LIN {X 0,Y 441.161,Z 147.091,A -85,B 0,C 180,E1 16742.338,E2 16742.338} C_VEL
LIN {X 0,Y 441.166,Z 147.092,A -85,B 0,C 180,E1 16738.571,E2 16738.571} C_VEL
LIN {X 0,Y 441.182,Z 147.089,A -85,B 0,C 180,E1 16734.929,E2 16734.929} C_VEL
LIN {X 0,Y 441.199,Z 147.088,A -85,B 0,C 180,E1 16731.266,E2 16731.266} C_VEL
LIN {X 0,Y 441.19,Z 147.092,A -85,B 0,C 180,E1 16727.434,E2 16727.434} C_VEL
LIN {X 0,Y 441.161,Z 147.096,A -85,B 0,C 180,E1 16723.813,E2 16723.813} C_VEL
LIN {X 0,Y 441.139,Z 147.048,A -85,B 0,C 180,E1 16720.124,E2 16720.124} C_VEL
LIN {X 0,Y 441.139,Z 147.074,A -85,B 0,C 180,E1 16716.348,E2 16716.348} C_VEL
LIN {X 0,Y 441.143,Z 147.081,A -85,B 0,C 180,E1 16712.606,E2 16712.606} C_VEL
LIN {X 0,Y 441.168,Z 147.048,A -85,B 0,C 180,E1 16709.038,E2 16709.038} C_VEL
LIN {X 0,Y 441.209,Z 147.301,A -85,B 0,C 180,E1 16705.273,E2 16705.273} C_VEL
LIN {X 0,Y 442.541,Z 150.696,A -85,B 0,C 180,E1 16704.503,E2 16704.503} C_VEL
LIN {X 0,Y 444.11,Z 153.026,A -85,B 0,C 180,E1 16703.923,E2 16703.923} C_VEL
LIN {X 0,Y 446.863,Z 158.227,A -85,B 0,C 180,E1 16702.8,E2 16702.8} C_VEL
LIN {X 0,Y 449.775,Z 163.654,A -85,B 0,C 180,E1 16701.667,E2 16701.667} C_VEL
LIN {X 0,Y 455.654,Z 174.722,A -85,B 0,C 180,E1 16699.494,E2 16699.494} C_VEL
LIN {X 0,Y 463.787,Z 191.79,A -85,B 0,C 180,E1 16696.55,E2 16696.55} C_VEL
LIN {X 0,Y 469.472,Z 204.192,A -85,B 0,C 180,E1 16694.656,E2 16694.656} C_VEL
LIN {X 0,Y 470.709,Z 206.682,A -85,B 0,C 180,E1 16694.44,E2 16694.44} C_VEL
LIN {X 0,Y 475.94,Z 241.296,A -85,B 0,C 180,E1 16693.055,E2 16693.055} C_VEL
LIN {X 0,Y 471.437,Z 427.319,A -85,B 0,C 180,E1 16689.939,E2 16689.939} C_VEL
LIN {X 0,Y 470.53,Z 435.022,A -85,B 0,C 180,E1 16689.894,E2 16689.894} C_VEL
LIN {X 0,Y 465.461,Z 455.605,A -85,B 0,C 180,E1 16690.074,E2 16690.074} C_VEL
LIN {X 0,Y 464.744,Z 462.217,A -85,B 0,C 180,E1 16690.028,E2 16690.028} C_VEL
LIN {X 0,Y 463.247,Z 517.307,A -85,B 0,C 180,E1 16689.082,E2 16689.082} C_VEL
LIN {X 0,Y 461.864,Z 538.343,A -85,B 0,C 180,E1 16688.519,E2 16688.519} C_VEL
LIN {X 0,Y 459.97,Z 559.929,A -85,B 0,C 180,E1 16687.719,E2 16687.719} C_VEL
LIN {X 0,Y 457.77,Z 579.888,A -85,B 0,C 180,E1 16686.759,E2 16686.759} C_VEL
LIN {X 0,Y 455.2,Z 599.112,A -85,B 0,C 180,E1 16685.596,E2 16685.596} C_VEL
LIN {X 0,Y 452.431,Z 617.858,A -85,B 0,C 180,E1 16684.223,E2 16684.223} C_VEL
LIN {X 0,Y 449.568,Z 634.992,A -85,B 0,C 180,E1 16682.713,E2 16682.713} C_VEL
LIN {X 0,Y 446.418,Z 652.781,A -85,B 0,C 180,E1 16680.856,E2 16680.856} C_VEL
LIN {X 0,Y 443.483,Z 669.165,A -85,B 0,C 180,E1 16678.846,E2 16678.846} C_VEL
LIN {X 0,Y 440.701,Z 684.442,A -85,B 0,C 180,E1 16676.632,E2 16676.632} C_VEL
LIN {X 0,Y 438.261,Z 698.588,A -85,B 0,C 180,E1 16674.245,E2 16674.245} C_VEL
LIN {X 0,Y 436.194,Z 711.687,A -85,B 0,C 180,E1 16671.656,E2 16671.656} C_VEL
LIN {X 0,Y 434.567,Z 723.315,A -85,B 0,C 180,E1 16668.93,E2 16668.93} C_VEL
LIN {X 0,Y 433.412,Z 732.998,A -85,B 0,C 180,E1 16666.208,E2 16666.208} C_VEL
LIN {X 0,Y 432.635,Z 741.395,A -85,B 0,C 180,E1 16663.351,E2 16663.351} C_VEL
LIN {X 0,Y 432.205,Z 748.037,A -85,B 0,C 180,E1 16660.519,E2 16660.519} C_VEL
LIN {X 0,Y 431.991,Z 753.036,A -85,B 0,C 180,E1 16657.715,E2 16657.715} C_VEL
LIN {X 0,Y 431.924,Z 756.563,A -85,B 0,C 180,E1 16654.913,E2 16654.913} C_VEL
LIN {X 0,Y 431.907,Z 758.422,A -85,B 0,C 180,E1 16652.255,E2 16652.255} C_VEL
LIN {X 0,Y 431.902,Z 758.898,A -85,B 0,C 180,E1 16649.337,E2 16649.337} C_VEL
LIN {X 0,Y 431.914,Z 757.928,A -85,B 0,C 180,E1 16646.682,E2 16646.682} C_VEL
LIN {X 0,Y 431.947,Z 755.334,A -85,B 0,C 180,E1 16643.888,E2 16643.888} C_VEL
LIN {X 0,Y 432.054,Z 751.256,A -85,B 0,C 180,E1 16641.08,E2 16641.08} C_VEL
LIN {X 0,Y 432.365,Z 745.257,A -85,B 0,C 180,E1 16638.123,E2 16638.123} C_VEL
LIN {X 0,Y 432.935,Z 737.852,A -85,B 0,C 180,E1 16635.283,E2 16635.283} C_VEL
LIN {X 0,Y 433.837,Z 729.193,A -85,B 0,C 180,E1 16632.566,E2 16632.566} C_VEL
LIN {X 0,Y 435.177,Z 718.684,A -85,B 0,C 180,E1 16629.841,E2 16629.841} C_VEL
LIN {X 0,Y 436.927,Z 706.823,A -85,B 0,C 180,E1 16627.249,E2 16627.249} C_VEL
LIN {X 0,Y 439.099,Z 693.731,A -85,B 0,C 180,E1 16624.799,E2 16624.799} C_VEL
LIN {X 0,Y 441.803,Z 678.428,A -85,B 0,C 180,E1 16622.359,E2 16622.359} C_VEL
LIN {X 0,Y 444.668,Z 662.439,A -85,B 0,C 180,E1 16620.204,E2 16620.204} C_VEL
LIN {X 0,Y 447.82,Z 645.002,A -85,B 0,C 180,E1 16618.203,E2 16618.203} C_VEL
LIN {X 0,Y 450.894,Z 627.379,A -85,B 0,C 180,E1 16616.486,E2 16616.486} C_VEL
LIN {X 0,Y 453.696,Z 609.476,A -85,B 0,C 180,E1 16615.042,E2 16615.042} C_VEL
LIN {X 0,Y 456.596,Z 589.037,A -85,B 0,C 180,E1 16613.678,E2 16613.678} C_VEL
LIN {X 0,Y 459.081,Z 568.729,A -85,B 0,C 180,E1 16612.581,E2 16612.581} C_VEL
LIN {X 0,Y 461.105,Z 547.553,A -85,B 0,C 180,E1 16611.7,E2 16611.7} C_VEL
LIN {X 0,Y 462.765,Z 525.423,A -85,B 0,C 180,E1 16611.024,E2 16611.024} C_VEL
LIN {X 0,Y 463.781,Z 503.548,A -85,B 0,C 180,E1 16610.568,E2 16610.568} C_VEL
LIN {X 0,Y 469.385,Z 276.561,A -85,B 0,C 180,E1 16606.757,E2 16606.757} C_VEL
LIN {X 0,Y 470.228,Z 241.192,A -85,B 0,C 180,E1 16606.129,E2 16606.129} C_VEL
LIN {X 0,Y 465.388,Z 210.155,A -85,B 0,C 180,E1 16604.831,E2 16604.831} C_VEL
LIN {X 0,Y 460.669,Z 202.535,A -85,B 0,C 180,E1 16603.991,E2 16603.991} C_VEL
LIN {X 0,Y 453.502,Z 187.149,A -85,B 0,C 180,E1 16601.409,E2 16601.409} C_VEL
LIN {X 0,Y 447.296,Z 174.728,A -85,B 0,C 180,E1 16599.077,E2 16599.077} C_VEL
LIN {X 0,Y 442.959,Z 166.509,A -85,B 0,C 180,E1 16597.387,E2 16597.387} C_VEL
LIN {X 0,Y 440.374,Z 161.697,A -85,B 0,C 180,E1 16596.341,E2 16596.341} C_VEL
LIN {X 0,Y 438.184,Z 157.597,A -85,B 0,C 180,E1 16595.421,E2 16595.421} C_VEL
LIN {X 0,Y 436.317,Z 154.259,A -85,B 0,C 180,E1 16594.633,E2 16594.633} C_VEL
LIN {X 0,Y 435.776,Z 153.005,A -85,B 0,C 180,E1 16594.363,E2 16594.363} C_VEL
LIN {X 0,Y 433.766,Z 150.233,A -85,B 0,C 180,E1 16593.588,E2 16593.588} C_VEL
LIN {X 0,Y 433.233,Z 148.247,A -85,B 0,C 180,E1 16593.097,E2 16593.097} C_VEL
LIN {X 0,Y 433.191,Z 148.054,A -85,B 0,C 180,E1 16589.525,E2 16589.525} C_VEL
LIN {X 0,Y 433.19,Z 148.038,A -85,B 0,C 180,E1 16585.717,E2 16585.717} C_VEL
LIN {X 0,Y 433.201,Z 148.086,A -85,B 0,C 180,E1 16581.903,E2 16581.903} C_VEL
LIN {X 0,Y 433.209,Z 148.039,A -85,B 0,C 180,E1 16578.155,E2 16578.155} C_VEL
LIN {X 0,Y 433.236,Z 148.069,A -85,B 0,C 180,E1 16574.433,E2 16574.433} C_VEL
LIN {X 0,Y 433.248,Z 148.069,A -85,B 0,C 180,E1 16570.639,E2 16570.639} C_VEL
LIN {X 0,Y 433.265,Z 148.068,A -85,B 0,C 180,E1 16566.759,E2 16566.759} C_VEL
LIN {X 0,Y 433.248,Z 148.072,A -85,B 0,C 180,E1 16562.91,E2 16562.91} C_VEL
LIN {X 0,Y 433.234,Z 148.075,A -85,B 0,C 180,E1 16559.207,E2 16559.207} C_VEL
LIN {X 0,Y 433.224,Z 148.079,A -85,B 0,C 180,E1 16555.5,E2 16555.5} C_VEL
LIN {X 0,Y 433.224,Z 148.08,A -85,B 0,C 180,E1 16551.773,E2 16551.773} C_VEL
LIN {X 0,Y 433.233,Z 148.08,A -85,B 0,C 180,E1 16548.012,E2 16548.012} C_VEL
LIN {X 0,Y 433.239,Z 148.026,A -85,B 0,C 180,E1 16544.228,E2 16544.228} C_VEL
LIN {X 0,Y 433.256,Z 148.061,A -85,B 0,C 180,E1 16540.45,E2 16540.45} C_VEL
LIN {X 0,Y 433.257,Z 148.052,A -85,B 0,C 180,E1 16536.613,E2 16536.613} C_VEL
LIN {X 0,Y 433.251,Z 148.032,A -85,B 0,C 180,E1 16532.81,E2 16532.81} C_VEL
LIN {X 0,Y 433.288,Z 148.284,A -85,B 0,C 180,E1 16529.184,E2 16529.184} C_VEL
LIN {X 0,Y 434.702,Z 151.729,A -85,B 0,C 180,E1 16528.371,E2 16528.371} C_VEL
LIN {X 0,Y 436.151,Z 153.411,A -85,B 0,C 180,E1 16527.87,E2 16527.87} C_VEL
LIN {X 0,Y 437.891,Z 157.074,A -85,B 0,C 180,E1 16527.082,E2 16527.082} C_VEL
LIN {X 0,Y 439.231,Z 159.208,A -85,B 0,C 180,E1 16526.573,E2 16526.573} C_VEL
LIN {X 0,Y 444.555,Z 168.866,A -85,B 0,C 180,E1 16524.504,E2 16524.504} C_VEL
LIN {X 0,Y 452.392,Z 179.593,A -85,B 0,C 180,E1 16522.928,E2 16522.928} C_VEL
LIN {X 0,Y 462.317,Z 193.566,A -85,B 0,C 180,E1 16521.134,E2 16521.134} C_VEL
LIN {X 0,Y 474.451,Z 211.926,A -85,B 0,C 180,E1 16519.09,E2 16519.09} C_VEL
LIN {X 0,Y 474.756,Z 213.111,A -85,B 0,C 180,E1 16519.025,E2 16519.025} C_VEL
LIN {X 0,Y 467.958,Z 425.301,A -85,B 0,C 180,E1 16515.184,E2 16515.184} C_VEL
LIN {X 0,Y 465.168,Z 512.028,A -85,B 0,C 180,E1 16513.602,E2 16513.602} C_VEL
LIN {X 0,Y 463.607,Z 534.936,A -85,B 0,C 180,E1 16512.987,E2 16512.987} C_VEL
LIN {X 0,Y 461.686,Z 557.609,A -85,B 0,C 180,E1 16512.17,E2 16512.17} C_VEL
LIN {X 0,Y 459.492,Z 578.606,A -85,B 0,C 180,E1 16511.197,E2 16511.197} C_VEL
LIN {X 0,Y 456.901,Z 600.642,A -85,B 0,C 180,E1 16509.961,E2 16509.961} C_VEL
LIN {X 0,Y 454.323,Z 620.398,A -85,B 0,C 180,E1 16508.623,E2 16508.623} C_VEL
LIN {X 0,Y 451.294,Z 641.976,A -85,B 0,C 180,E1 16506.888,E2 16506.888} C_VEL
LIN {X 0,Y 448.466,Z 660.864,A -85,B 0,C 180,E1 16505.113,E2 16505.113} C_VEL
LIN {X 0,Y 445.625,Z 678.963,A -85,B 0,C 180,E1 16503.116,E2 16503.116} C_VEL
LIN {X 0,Y 442.903,Z 696.137,A -85,B 0,C 180,E1 16500.924,E2 16500.924} C_VEL
LIN {X 0,Y 440.427,Z 711.612,A -85,B 0,C 180,E1 16498.62,E2 16498.62} C_VEL
LIN {X 0,Y 438.093,Z 726.942,A -85,B 0,C 180,E1 16495.988,E2 16495.988} C_VEL
LIN {X 0,Y 436.406,Z 738.708,A -85,B 0,C 180,E1 16493.637,E2 16493.637} C_VEL
LIN {X 0,Y 434.67,Z 751.426,A -85,B 0,C 180,E1 16490.576,E2 16490.576} C_VEL
LIN {X 0,Y 433.525,Z 761.436,A -85,B 0,C 180,E1 16487.724,E2 16487.724} C_VEL
LIN {X 0,Y 432.749,Z 769.699,A -85,B 0,C 180,E1 16484.86,E2 16484.86} C_VEL
LIN {X 0,Y 432.293,Z 776.47,A -85,B 0,C 180,E1 16482.014,E2 16482.014} C_VEL
LIN {X 0,Y 432.033,Z 781.843,A -85,B 0,C 180,E1 16479.054,E2 16479.054} C_VEL
LIN {X 0,Y 431.943,Z 785.438,A -85,B 0,C 180,E1 16476.379,E2 16476.379} C_VEL
LIN {X 0,Y 431.91,Z 787.984,A -85,B 0,C 180,E1 16473.318,E2 16473.318} C_VEL
LIN {X 0,Y 431.901,Z 788.894,A -85,B 0,C 180,E1 16470.663,E2 16470.663} C_VEL
LIN {X 0,Y 431.907,Z 788.46,A -85,B 0,C 180,E1 16467.612,E2 16467.612} C_VEL
LIN {X 0,Y 431.919,Z 786.727,A -85,B 0,C 180,E1 16464.953,E2 16464.953} C_VEL
LIN {X 0,Y 431.998,Z 783.494,A -85,B 0,C 180,E1 16462.018,E2 16462.018} C_VEL
LIN {X 0,Y 432.177,Z 778.573,A -85,B 0,C 180,E1 16459.064,E2 16459.064} C_VEL
LIN {X 0,Y 432.574,Z 772.169,A -85,B 0,C 180,E1 16456.091,E2 16456.091} C_VEL
LIN {X 0,Y 433.216,Z 764.337,A -85,B 0,C 180,E1 16453.232,E2 16453.232} C_VEL
LIN {X 0,Y 434.298,Z 754.411,A -85,B 0,C 180,E1 16450.219,E2 16450.219} C_VEL
LIN {X 0,Y 435.626,Z 744.143,A -85,B 0,C 180,E1 16447.605,E2 16447.605} C_VEL
LIN {X 0,Y 437.263,Z 732.76,A -85,B 0,C 180,E1 16445.119,E2 16445.119} C_VEL
LIN {X 0,Y 439.298,Z 718.902,A -85,B 0,C 180,E1 16442.579,E2 16442.579} C_VEL
LIN {X 0,Y 441.866,Z 702.557,A -85,B 0,C 180,E1 16439.996,E2 16439.996} C_VEL
LIN {X 0,Y 444.462,Z 686.329,A -85,B 0,C 180,E1 16437.782,E2 16437.782} C_VEL
LIN {X 0,Y 447.256,Z 668.628,A -85,B 0,C 180,E1 16435.713,E2 16435.713} C_VEL
LIN {X 0,Y 450.17,Z 649.602,A -85,B 0,C 180,E1 16433.787,E2 16433.787} C_VEL
LIN {X 0,Y 453.07,Z 629.567,A -85,B 0,C 180,E1 16432.078,E2 16432.078} C_VEL
LIN {X 0,Y 455.981,Z 608.032,A -85,B 0,C 180,E1 16430.514,E2 16430.514} C_VEL
LIN {X 0,Y 458.414,Z 587.979,A -85,B 0,C 180,E1 16429.297,E2 16429.297} C_VEL
LIN {X 0,Y 460.893,Z 565.197,A -85,B 0,C 180,E1 16428.159,E2 16428.159} C_VEL
LIN {X 0,Y 463.018,Z 542.927,A -85,B 0,C 180,E1 16427.272,E2 16427.272} C_VEL
LIN {X 0,Y 464.644,Z 520.593,A -85,B 0,C 180,E1 16426.609,E2 16426.609} C_VEL
LIN {X 0,Y 465.814,Z 496.635,A -85,B 0,C 180,E1 16426.095,E2 16426.095} C_VEL
LIN {X 0,Y 472.407,Z 285.373,A -85,B 0,C 180,E1 16422.285,E2 16422.285} C_VEL
LIN {X 0,Y 474.674,Z 212.296,A -85,B 0,C 180,E1 16420.946,E2 16420.946} C_VEL
LIN {X 0,Y 462.586,Z 193.972,A -85,B 0,C 180,E1 16418.917,E2 16418.917} C_VEL
LIN {X 0,Y 452.787,Z 180.133,A -85,B 0,C 180,E1 16417.153,E2 16417.153} C_VEL
LIN {X 0,Y 444.836,Z 169.404,A -85,B 0,C 180,E1 16415.602,E2 16415.602} C_VEL
LIN {X 0,Y 440.788,Z 162.144,A -85,B 0,C 180,E1 16414.075,E2 16414.075} C_VEL
LIN {X 0,Y 438.217,Z 157.492,A -85,B 0,C 180,E1 16413.046,E2 16413.046} C_VEL
LIN {X 0,Y 436.356,Z 154.067,A -85,B 0,C 180,E1 16412.269,E2 16412.269} C_VEL
LIN {X 0,Y 433.528,Z 149.347,A -85,B 0,C 180,E1 16411.105,E2 16411.105} C_VEL
LIN {X 0,Y 433.259,Z 148.113,A -85,B 0,C 180,E1 16410.713,E2 16410.713} C_VEL
LIN {X 0,Y 433.249,Z 148.033,A -85,B 0,C 180,E1 16406.893,E2 16406.893} C_VEL
LIN {X 0,Y 433.258,Z 148.045,A -85,B 0,C 180,E1 16403.099,E2 16403.099} C_VEL
LIN {X 0,Y 433.26,Z 148.07,A -85,B 0,C 180,E1 16399.269,E2 16399.269} C_VEL
LIN {X 0,Y 433.256,Z 148.022,A -85,B 0,C 180,E1 16395.39,E2 16395.39} C_VEL
LIN {X 0,Y 433.253,Z 148.077,A -85,B 0,C 180,E1 16391.582,E2 16391.582} C_VEL
LIN {X 0,Y 433.239,Z 148.075,A -85,B 0,C 180,E1 16387.826,E2 16387.826} C_VEL
LIN {X 0,Y 433.225,Z 148.075,A -85,B 0,C 180,E1 16384.103,E2 16384.103} C_VEL
LIN {X 0,Y 433.221,Z 148.073,A -85,B 0,C 180,E1 16380.397,E2 16380.397} C_VEL
LIN {X 0,Y 433.229,Z 148.07,A -85,B 0,C 180,E1 16376.692,E2 16376.692} C_VEL
LIN {X 0,Y 433.242,Z 148.069,A -85,B 0,C 180,E1 16372.908,E2 16372.908} C_VEL
LIN {X 0,Y 433.252,Z 148.068,A -85,B 0,C 180,E1 16369.226,E2 16369.226} C_VEL
LIN {X 0,Y 433.251,Z 148.068,A -85,B 0,C 180,E1 16365.431,E2 16365.431} C_VEL
LIN {X 0,Y 433.221,Z 148.037,A -85,B 0,C 180,E1 16361.706,E2 16361.706} C_VEL
LIN {X 0,Y 433.206,Z 148.085,A -85,B 0,C 180,E1 16358.043,E2 16358.043} C_VEL
LIN {X 0,Y 433.194,Z 148.036,A -85,B 0,C 180,E1 16354.283,E2 16354.283} C_VEL
LIN {X 0,Y 433.2,Z 148.057,A -85,B 0,C 180,E1 16350.553,E2 16350.553} C_VEL
LIN {X 0,Y 433.222,Z 148.116,A -85,B 0,C 180,E1 16346.874,E2 16346.874} C_VEL
LIN {X 0,Y 433.388,Z 149.085,A -85,B 0,C 180,E1 16346.537,E2 16346.537} C_VEL
LIN {X 0,Y 435.142,Z 152.362,A -85,B 0,C 180,E1 16345.739,E2 16345.739} C_VEL
LIN {X 0,Y 436.163,Z 153.761,A -85,B 0,C 180,E1 16345.353,E2 16345.353} C_VEL
LIN {X 0,Y 437.94,Z 157.295,A -85,B 0,C 180,E1 16344.556,E2 16344.556} C_VEL
LIN {X 0,Y 439.216,Z 159.548,A -85,B 0,C 180,E1 16344.032,E2 16344.032} C_VEL
LIN {X 0,Y 441.768,Z 164.304,A -85,B 0,C 180,E1 16342.984,E2 16342.984} C_VEL
LIN {X 0,Y 446.266,Z 172.624,A -85,B 0,C 180,E1 16341.23,E2 16341.23} C_VEL
LIN {X 0,Y 453.287,Z 186.751,A -85,B 0,C 180,E1 16338.567,E2 16338.567} C_VEL
LIN {X 0,Y 460.637,Z 202.485,A -85,B 0,C 180,E1 16335.926,E2 16335.926} C_VEL
LIN {X 0,Y 465.613,Z 210.899,A -85,B 0,C 180,E1 16335.028,E2 16335.028} C_VEL
LIN {X 0,Y 470.323,Z 242.898,A -85,B 0,C 180,E1 16333.727,E2 16333.727} C_VEL
LIN {X 0,Y 464.744,Z 462.217,A -85,B 0,C 180,E1 16330.028,E2 16330.028} C_VEL
LIN {X 0,Y 463.827,Z 469.919,A -85,B 0,C 180,E1 16329.984,E2 16329.984} C_VEL
LIN {X 0,Y 458.762,Z 490.496,A -85,B 0,C 180,E1 16330.168,E2 16330.168} C_VEL
LIN {X 0,Y 458.025,Z 497.107,A -85,B 0,C 180,E1 16330.124,E2 16330.124} C_VEL
LIN {X 0,Y 456.967,Z 522.832,A -85,B 0,C 180,E1 16329.621,E2 16329.621} C_VEL
LIN {X 0,Y 455.467,Z 543.801,A -85,B 0,C 180,E1 16329.015,E2 16329.015} C_VEL
LIN {X 0,Y 453.441,Z 564.036,A -85,B 0,C 180,E1 16328.206,E2 16328.206} C_VEL
LIN {X 0,Y 450.829,Z 585.53,A -85,B 0,C 180,E1 16327.102,E2 16327.102} C_VEL
LIN {X 0,Y 448.092,Z 605.047,A -85,B 0,C 180,E1 16325.854,E2 16325.854} C_VEL
LIN {X 0,Y 445.052,Z 623.573,A -85,B 0,C 180,E1 16324.403,E2 16324.403} C_VEL
LIN {X 0,Y 441.663,Z 642.761,A -85,B 0,C 180,E1 16322.601,E2 16322.601} C_VEL
LIN {X 0,Y 438.558,Z 659.443,A -85,B 0,C 180,E1 16320.738,E2 16320.738} C_VEL
LIN {X 0,Y 435.401,Z 675.439,A -85,B 0,C 180,E1 16318.606,E2 16318.606} C_VEL
LIN {X 0,Y 432.452,Z 690.789,A -85,B 0,C 180,E1 16316.206,E2 16316.206} C_VEL
LIN {X 0,Y 429.989,Z 704.362,A -85,B 0,C 180,E1 16313.72,E2 16313.72} C_VEL
LIN {X 0,Y 427.956,Z 716.558,A -85,B 0,C 180,E1 16311.087,E2 16311.087} C_VEL
LIN {X 0,Y 426.364,Z 727.38,A -85,B 0,C 180,E1 16308.314,E2 16308.314} C_VEL
LIN {X 0,Y 425.227,Z 736.836,A -85,B 0,C 180,E1 16305.408,E2 16305.408} C_VEL
LIN {X 0,Y 424.52,Z 744.496,A -85,B 0,C 180,E1 16302.514,E2 16302.514} C_VEL
LIN {X 0,Y 424.139,Z 750.39,A -85,B 0,C 180,E1 16299.635,E2 16299.635} C_VEL
LIN {X 0,Y 423.971,Z 754.919,A -85,B 0,C 180,E1 16296.636,E2 16296.636} C_VEL
LIN {X 0,Y 423.918,Z 757.597,A -85,B 0,C 180,E1 16293.889,E2 16293.889} C_VEL
LIN {X 0,Y 423.909,Z 758.895,A -85,B 0,C 180,E1 16290.946,E2 16290.946} C_VEL
LIN {X 0,Y 423.908,Z 758.739,A -85,B 0,C 180,E1 16288.108,E2 16288.108} C_VEL
LIN {X 0,Y 423.925,Z 756.98,A -85,B 0,C 180,E1 16285.265,E2 16285.265} C_VEL
LIN {X 0,Y 423.997,Z 753.593,A -85,B 0,C 180,E1 16282.275,E2 16282.275} C_VEL
LIN {X 0,Y 424.23,Z 748.821,A -85,B 0,C 180,E1 16279.407,E2 16279.407} C_VEL
LIN {X 0,Y 424.7,Z 742.233,A -85,B 0,C 180,E1 16276.487,E2 16276.487} C_VEL
LIN {X 0,Y 425.582,Z 733.601,A -85,B 0,C 180,E1 16273.447,E2 16273.447} C_VEL
LIN {X 0,Y 426.821,Z 724.199,A -85,B 0,C 180,E1 16270.713,E2 16270.713} C_VEL
LIN {X 0,Y 428.567,Z 712.668,A -85,B 0,C 180,E1 16267.938,E2 16267.938} C_VEL
LIN {X 0,Y 430.784,Z 699.747,A -85,B 0,C 180,E1 16265.306,E2 16265.306} C_VEL
LIN {X 0,Y 433.468,Z 685.485,A -85,B 0,C 180,E1 16262.825,E2 16262.825} C_VEL
LIN {X 0,Y 436.448,Z 670.221,A -85,B 0,C 180,E1 16260.568,E2 16260.568} C_VEL
LIN {X 0,Y 439.538,Z 654.095,A -85,B 0,C 180,E1 16258.545,E2 16258.545} C_VEL
LIN {X 0,Y 442.751,Z 636.918,A -85,B 0,C 180,E1 16256.719,E2 16256.719} C_VEL
LIN {X 0,Y 445.701,Z 619.815,A -85,B 0,C 180,E1 16255.191,E2 16255.191} C_VEL
LIN {X 0,Y 448.767,Z 600.196,A -85,B 0,C 180,E1 16253.726,E2 16253.726} C_VEL
LIN {X 0,Y 451.59,Z 580.024,A -85,B 0,C 180,E1 16252.493,E2 16252.493} C_VEL
LIN {X 0,Y 453.833,Z 560.576,A -85,B 0,C 180,E1 16251.551,E2 16251.551} C_VEL
LIN {X 0,Y 455.843,Z 538.851,A -85,B 0,C 180,E1 16250.734,E2 16250.734} C_VEL
LIN {X 0,Y 457.3,Z 517.7,A -85,B 0,C 180,E1 16250.163,E2 16250.163} C_VEL
LIN {X 0,Y 458.75,Z 468.357,A -85,B 0,C 180,E1 16249.302,E2 16249.302} C_VEL
LIN {X 0,Y 464.821,Z 243.745,A -85,B 0,C 180,E1 16245.477,E2 16245.477} C_VEL
LIN {X 0,Y 460.395,Z 214.629,A -85,B 0,C 180,E1 16244.241,E2 16244.241} C_VEL
LIN {X 0,Y 452.254,Z 201.732,A -85,B 0,C 180,E1 16242.744,E2 16242.744} C_VEL
LIN {X 0,Y 444.626,Z 185.556,A -85,B 0,C 180,E1 16239.859,E2 16239.859} C_VEL
LIN {X 0,Y 437.958,Z 172.638,A -85,B 0,C 180,E1 16237.229,E2 16237.229} C_VEL
LIN {X 0,Y 432.871,Z 163.274,A -85,B 0,C 180,E1 16235.11,E2 16235.11} C_VEL
LIN {X 0,Y 430.457,Z 158.802,A -85,B 0,C 180,E1 16234.042,E2 16234.042} C_VEL
LIN {X 0,Y 428.362,Z 155.116,A -85,B 0,C 180,E1 16233.106,E2 16233.106} C_VEL
LIN {X 0,Y 427.468,Z 153.606,A -85,B 0,C 180,E1 16232.705,E2 16232.705} C_VEL
LIN {X 0,Y 425.661,Z 150.765,A -85,B 0,C 180,E1 16231.905,E2 16231.905} C_VEL
LIN {X 0,Y 425.269,Z 149.186,A -85,B 0,C 180,E1 16231.463,E2 16231.463} C_VEL
LIN {X 0,Y 425.254,Z 149.07,A -85,B 0,C 180,E1 16227.745,E2 16227.745} C_VEL
LIN {X 0,Y 425.256,Z 149.039,A -85,B 0,C 180,E1 16223.853,E2 16223.853} C_VEL
LIN {X 0,Y 425.273,Z 149.025,A -85,B 0,C 180,E1 16220.219,E2 16220.219} C_VEL
LIN {X 0,Y 425.296,Z 149.067,A -85,B 0,C 180,E1 16216.43,E2 16216.43} C_VEL
LIN {X 0,Y 425.314,Z 149.071,A -85,B 0,C 180,E1 16212.687,E2 16212.687} C_VEL
LIN {X 0,Y 425.317,Z 149.068,A -85,B 0,C 180,E1 16208.79,E2 16208.79} C_VEL
LIN {X 0,Y 425.306,Z 149.065,A -85,B 0,C 180,E1 16204.99,E2 16204.99} C_VEL
LIN {X 0,Y 425.293,Z 149.065,A -85,B 0,C 180,E1 16201.213,E2 16201.213} C_VEL
LIN {X 0,Y 425.286,Z 149.064,A -85,B 0,C 180,E1 16197.44,E2 16197.44} C_VEL
LIN {X 0,Y 425.283,Z 149.061,A -85,B 0,C 180,E1 16193.656,E2 16193.656} C_VEL
LIN {X 0,Y 425.287,Z 149.056,A -85,B 0,C 180,E1 16189.844,E2 16189.844} C_VEL
LIN {X 0,Y 425.295,Z 149.028,A -85,B 0,C 180,E1 16186.126,E2 16186.126} C_VEL
LIN {X 0,Y 425.312,Z 149.052,A -85,B 0,C 180,E1 16182.346,E2 16182.346} C_VEL
LIN {X 0,Y 425.317,Z 149.013,A -85,B 0,C 180,E1 16178.486,E2 16178.486} C_VEL
LIN {X 0,Y 425.319,Z 149.048,A -85,B 0,C 180,E1 16174.669,E2 16174.669} C_VEL
LIN {X 0,Y 425.327,Z 149.122,A -85,B 0,C 180,E1 16170.882,E2 16170.882} C_VEL
LIN {X 0,Y 425.688,Z 150.647,A -85,B 0,C 180,E1 16170.446,E2 16170.446} C_VEL
LIN {X 0,Y 427.469,Z 153.609,A -85,B 0,C 180,E1 16169.654,E2 16169.654} C_VEL
LIN {X 0,Y 428.457,Z 154.941,A -85,B 0,C 180,E1 16169.265,E2 16169.265} C_VEL
LIN {X 0,Y 430.529,Z 158.747,A -85,B 0,C 180,E1 16168.341,E2 16168.341} C_VEL
LIN {X 0,Y 431.741,Z 160.97,A -85,B 0,C 180,E1 16167.816,E2 16167.816} C_VEL
LIN {X 0,Y 434.29,Z 165.382,A -85,B 0,C 180,E1 16166.774,E2 16166.774} C_VEL
LIN {X 0,Y 437.352,Z 170.801,A -85,B 0,C 180,E1 16165.617,E2 16165.617} C_VEL
LIN {X 0,Y 448.036,Z 184.976,A -85,B 0,C 180,E1 16163.467,E2 16163.467} C_VEL
LIN {X 0,Y 458.401,Z 199.726,A -85,B 0,C 180,E1 16161.542,E2 16161.542} C_VEL
LIN {X 0,Y 469.156,Z 216.172,A -85,B 0,C 180,E1 16159.679,E2 16159.679} C_VEL
LIN {X 0,Y 461.958,Z 428.692,A -85,B 0,C 180,E1 16155.794,E2 16155.794} C_VEL
LIN {X 0,Y 459.104,Z 512.038,A -85,B 0,C 180,E1 16154.252,E2 16154.252} C_VEL
LIN {X 0,Y 457.44,Z 535.074,A -85,B 0,C 180,E1 16153.627,E2 16153.627} C_VEL
LIN {X 0,Y 455.413,Z 557.626,A -85,B 0,C 180,E1 16152.804,E2 16152.804} C_VEL
LIN {X 0,Y 453.114,Z 578.291,A -85,B 0,C 180,E1 16151.831,E2 16151.831} C_VEL
LIN {X 0,Y 450.343,Z 600.169,A -85,B 0,C 180,E1 16150.58,E2 16150.58} C_VEL
LIN {X 0,Y 447.307,Z 621.903,A -85,B 0,C 180,E1 16149.075,E2 16149.075} C_VEL
LIN {X 0,Y 444.264,Z 642.301,A -85,B 0,C 180,E1 16147.396,E2 16147.396} C_VEL
LIN {X 0,Y 441.254,Z 661.469,A -85,B 0,C 180,E1 16145.563,E2 16145.563} C_VEL
LIN {X 0,Y 438.232,Z 679.645,A -85,B 0,C 180,E1 16143.513,E2 16143.513} C_VEL
LIN {X 0,Y 435.27,Z 697.51,A -85,B 0,C 180,E1 16141.184,E2 16141.184} C_VEL
LIN {X 0,Y 432.875,Z 711.788,A -85,B 0,C 180,E1 16139.015,E2 16139.015} C_VEL
LIN {X 0,Y 430.346,Z 727.478,A -85,B 0,C 180,E1 16136.257,E2 16136.257} C_VEL
LIN {X 0,Y 428.458,Z 740.151,A -85,B 0,C 180,E1 16133.664,E2 16133.664} C_VEL
LIN {X 0,Y 426.846,Z 751.896,A -85,B 0,C 180,E1 16130.832,E2 16130.832} C_VEL
LIN {X 0,Y 425.672,Z 761.435,A -85,B 0,C 180,E1 16128.062,E2 16128.062} C_VEL
LIN {X 0,Y 424.833,Z 769.698,A -85,B 0,C 180,E1 16125.143,E2 16125.143} C_VEL
LIN {X 0,Y 424.33,Z 776.469,A -85,B 0,C 180,E1 16122.243,E2 16122.243} C_VEL
LIN {X 0,Y 424.05,Z 781.843,A -85,B 0,C 180,E1 16119.226,E2 16119.226} C_VEL
LIN {X 0,Y 423.948,Z 785.438,A -85,B 0,C 180,E1 16116.5,E2 16116.5} C_VEL
LIN {X 0,Y 423.91,Z 787.984,A -85,B 0,C 180,E1 16113.38,E2 16113.38} C_VEL
LIN {X 0,Y 423.901,Z 788.894,A -85,B 0,C 180,E1 16110.676,E2 16110.676} C_VEL
LIN {X 0,Y 423.907,Z 788.46,A -85,B 0,C 180,E1 16107.567,E2 16107.567} C_VEL
LIN {X 0,Y 423.921,Z 786.727,A -85,B 0,C 180,E1 16104.858,E2 16104.858} C_VEL
LIN {X 0,Y 424.004,Z 783.495,A -85,B 0,C 180,E1 16101.866,E2 16101.866} C_VEL
LIN {X 0,Y 424.203,Z 778.573,A -85,B 0,C 180,E1 16098.856,E2 16098.856} C_VEL
LIN {X 0,Y 424.636,Z 772.168,A -85,B 0,C 180,E1 16095.826,E2 16095.826} C_VEL
LIN {X 0,Y 425.343,Z 764.336,A -85,B 0,C 180,E1 16092.913,E2 16092.913} C_VEL
LIN {X 0,Y 426.524,Z 754.41,A -85,B 0,C 180,E1 16089.843,E2 16089.843} C_VEL
LIN {X 0,Y 427.832,Z 744.431,A -85,B 0,C 180,E1 16087.319,E2 16087.319} C_VEL
LIN {X 0,Y 429.744,Z 731.43,A -85,B 0,C 180,E1 16084.506,E2 16084.506} C_VEL
LIN {X 0,Y 431.909,Z 717.707,A -85,B 0,C 180,E1 16081.97,E2 16081.97} C_VEL
LIN {X 0,Y 434.631,Z 701.255,A -85,B 0,C 180,E1 16079.359,E2 16079.359} C_VEL
LIN {X 0,Y 437.361,Z 685.095,A -85,B 0,C 180,E1 16077.15,E2 16077.15} C_VEL
LIN {X 0,Y 440.332,Z 666.905,A -85,B 0,C 180,E1 16075.025,E2 16075.025} C_VEL
LIN {X 0,Y 443.444,Z 647.623,A -85,B 0,C 180,E1 16073.081,E2 16073.081} C_VEL
LIN {X 0,Y 446.397,Z 628.2,A -85,B 0,C 180,E1 16071.417,E2 16071.417} C_VEL
LIN {X 0,Y 449.616,Z 605.374,A -85,B 0,C 180,E1 16069.76,E2 16069.76} C_VEL
LIN {X 0,Y 452.422,Z 584.185,A -85,B 0,C 180,E1 16068.472,E2 16068.472} C_VEL
LIN {X 0,Y 454.84,Z 562.845,A -85,B 0,C 180,E1 16067.427,E2 16067.427} C_VEL
LIN {X 0,Y 457.051,Z 540.316,A -85,B 0,C 180,E1 16066.542,E2 16066.542} C_VEL
LIN {X 0,Y 458.666,Z 518.801,A -85,B 0,C 180,E1 16065.916,E2 16065.916} C_VEL
LIN {X 0,Y 459.971,Z 490.545,A -85,B 0,C 180,E1 16065.331,E2 16065.331} C_VEL
LIN {X 0,Y 466.934,Z 280.725,A -85,B 0,C 180,E1 16061.501,E2 16061.501} C_VEL
LIN {X 0,Y 469.017,Z 215.875,A -85,B 0,C 180,E1 16060.296,E2 16060.296} C_VEL
LIN {X 0,Y 456.309,Z 196.625,A -85,B 0,C 180,E1 16058.084,E2 16058.084} C_VEL
LIN {X 0,Y 443.751,Z 179.08,A -85,B 0,C 180,E1 16055.702,E2 16055.702} C_VEL
LIN {X 0,Y 436.88,Z 170.001,A -85,B 0,C 180,E1 16054.264,E2 16054.264} C_VEL
LIN {X 0,Y 433.307,Z 163.618,A -85,B 0,C 180,E1 16052.838,E2 16052.838} C_VEL
LIN {X 0,Y 430.485,Z 158.697,A -85,B 0,C 180,E1 16051.662,E2 16051.662} C_VEL
LIN {X 0,Y 428.427,Z 154.85,A -85,B 0,C 180,E1 16050.737,E2 16050.737} C_VEL
LIN {X 0,Y 425.886,Z 151.18,A -85,B 0,C 180,E1 16049.694,E2 16049.694} C_VEL
LIN {X 0,Y 425.37,Z 149.409,A -85,B 0,C 180,E1 16049.269,E2 16049.269} C_VEL
LIN {X 0,Y 425.298,Z 149.026,A -85,B 0,C 180,E1 16048.166,E2 16048.166} C_VEL
LIN {X 0,Y 425.301,Z 149.072,A -85,B 0,C 180,E1 16044.294,E2 16044.294} C_VEL
LIN {X 0,Y 425.295,Z 149.025,A -85,B 0,C 180,E1 16040.505,E2 16040.505} C_VEL
LIN {X 0,Y 425.305,Z 149.028,A -85,B 0,C 180,E1 16036.808,E2 16036.808} C_VEL
LIN {X 0,Y 425.317,Z 149.05,A -85,B 0,C 180,E1 16033.043,E2 16033.043} C_VEL
LIN {X 0,Y 425.32,Z 149.062,A -85,B 0,C 180,E1 16029.133,E2 16029.133} C_VEL
LIN {X 0,Y 425.32,Z 149.068,A -85,B 0,C 180,E1 16025.26,E2 16025.26} C_VEL
LIN {X 0,Y 425.322,Z 149.07,A -85,B 0,C 180,E1 16021.347,E2 16021.347} C_VEL
LIN {X 0,Y 425.308,Z 149.07,A -85,B 0,C 180,E1 16017.575,E2 16017.575} C_VEL
LIN {X 0,Y 425.292,Z 149.069,A -85,B 0,C 180,E1 16013.791,E2 16013.791} C_VEL
LIN {X 0,Y 425.276,Z 149.068,A -85,B 0,C 180,E1 16010.088,E2 16010.088} C_VEL
LIN {X 0,Y 425.269,Z 149.063,A -85,B 0,C 180,E1 16006.263,E2 16006.263} C_VEL
LIN {X 0,Y 425.269,Z 149.042,A -85,B 0,C 180,E1 16002.486,E2 16002.486} C_VEL
LIN {X 0,Y 425.279,Z 149.047,A -85,B 0,C 180,E1 15998.773,E2 15998.773} C_VEL
LIN {X 0,Y 425.299,Z 149.019,A -85,B 0,C 180,E1 15995.113,E2 15995.113} C_VEL
LIN {X 0,Y 425.31,Z 149.056,A -85,B 0,C 180,E1 15991.188,E2 15991.188} C_VEL
LIN {X 0,Y 425.286,Z 149.278,A -85,B 0,C 180,E1 15988.38,E2 15988.38} C_VEL
LIN {X 0,Y 426.564,Z 152.488,A -85,B 0,C 180,E1 15987.536,E2 15987.536} C_VEL
LIN {X 0,Y 428.217,Z 154.615,A -85,B 0,C 180,E1 15986.881,E2 15986.881} C_VEL
LIN {X 0,Y 429.865,Z 158.077,A -85,B 0,C 180,E1 15986.066,E2 15986.066} C_VEL
LIN {X 0,Y 431.173,Z 160.024,A -85,B 0,C 180,E1 15985.541,E2 15985.541} C_VEL
LIN {X 0,Y 436.454,Z 169.84,A -85,B 0,C 180,E1 15983.279,E2 15983.279} C_VEL
LIN {X 0,Y 443.062,Z 182.448,A -85,B 0,C 180,E1 15980.644,E2 15980.644} C_VEL
LIN {X 0,Y 450.639,Z 198.162,A -85,B 0,C 180,E1 15977.756,E2 15977.756} C_VEL
LIN {X 0,Y 452.976,Z 203.077,A -85,B 0,C 180,E1 15976.995,E2 15976.995} C_VEL
LIN {X 0,Y 460.606,Z 215.289,A -85,B 0,C 180,E1 15975.619,E2 15975.619} C_VEL
LIN {X 0,Y 464.77,Z 244.555,A -85,B 0,C 180,E1 15974.415,E2 15974.415} C_VEL
LIN {X 0,Y 458.632,Z 472.586,A -85,B 0,C 180,E1 15970.536,E2 15970.536} C_VEL
LIN {X 0,Y 458.025,Z 497.107,A -85,B 0,C 180,E1 15970.124,E2 15970.124} C_VEL
LIN {X 0,Y 457.061,Z 504.813,A -85,B 0,C 180,E1 15970.082,E2 15970.082} C_VEL
LIN {X 0,Y 451.788,Z 524.21,A -85,B 0,C 180,E1 15970.199,E2 15970.199} C_VEL
LIN {X 0,Y 450.465,Z 531.785,A -85,B 0,C 180,E1 15970.079,E2 15970.079} C_VEL
LIN {X 0,Y 448.585,Z 552.863,A -85,B 0,C 180,E1 15969.364,E2 15969.364} C_VEL
LIN {X 0,Y 446.285,Z 573.329,A -85,B 0,C 180,E1 15968.44,E2 15968.44} C_VEL
LIN {X 0,Y 443.61,Z 593.175,A -85,B 0,C 180,E1 15967.321,E2 15967.321} C_VEL
LIN {X 0,Y 440.592,Z 612.071,A -85,B 0,C 180,E1 15965.997,E2 15965.997} C_VEL
LIN {X 0,Y 437.159,Z 631.657,A -85,B 0,C 180,E1 15964.343,E2 15964.343} C_VEL
LIN {X 0,Y 433.817,Z 649.448,A -85,B 0,C 180,E1 15962.548,E2 15962.548} C_VEL
LIN {X 0,Y 430.498,Z 665.826,A -85,B 0,C 180,E1 15960.572,E2 15960.572} C_VEL
LIN {X 0,Y 427.306,Z 681.419,A -85,B 0,C 180,E1 15958.359,E2 15958.359} C_VEL
LIN {X 0,Y 424.427,Z 695.625,A -85,B 0,C 180,E1 15955.987,E2 15955.987} C_VEL
LIN {X 0,Y 421.795,Z 709.082,A -85,B 0,C 180,E1 15953.32,E2 15953.32} C_VEL
LIN {X 0,Y 419.683,Z 721.104,A -85,B 0,C 180,E1 15950.5,E2 15950.5} C_VEL
LIN {X 0,Y 418.159,Z 731.274,A -85,B 0,C 180,E1 15947.678,E2 15947.678} C_VEL
LIN {X 0,Y 417.082,Z 740.011,A -85,B 0,C 180,E1 15944.72,E2 15944.72} C_VEL
LIN {X 0,Y 416.43,Z 746.976,A -85,B 0,C 180,E1 15941.776,E2 15941.776} C_VEL
LIN {X 0,Y 416.093,Z 752.389,A -85,B 0,C 180,E1 15938.846,E2 15938.846} C_VEL
LIN {X 0,Y 415.962,Z 756.164,A -85,B 0,C 180,E1 15935.933,E2 15935.933} C_VEL
LIN {X 0,Y 415.916,Z 758.526,A -85,B 0,C 180,E1 15932.894,E2 15932.894} C_VEL
LIN {X 0,Y 415.918,Z 759.343,A -85,B 0,C 180,E1 15930,E2 15930} C_VEL
LIN {X 0,Y 415.916,Z 758.569,A -85,B 0,C 180,E1 15927.106,E2 15927.106} C_VEL
LIN {X 0,Y 415.955,Z 756.419,A -85,B 0,C 180,E1 15924.206,E2 15924.206} C_VEL
LIN {X 0,Y 416.068,Z 752.916,A -85,B 0,C 180,E1 15921.432,E2 15921.432} C_VEL
LIN {X 0,Y 416.396,Z 747.455,A -85,B 0,C 180,E1 15918.364,E2 15918.364} C_VEL
LIN {X 0,Y 417.024,Z 740.648,A -85,B 0,C 180,E1 15915.419,E2 15915.419} C_VEL
LIN {X 0,Y 418.052,Z 731.984,A -85,B 0,C 180,E1 15912.462,E2 15912.462} C_VEL
LIN {X 0,Y 419.537,Z 721.989,A -85,B 0,C 180,E1 15909.638,E2 15909.638} C_VEL
LIN {X 0,Y 421.498,Z 710.82,A -85,B 0,C 180,E1 15906.959,E2 15906.959} C_VEL
LIN {X 0,Y 424.027,Z 697.559,A -85,B 0,C 180,E1 15904.287,E2 15904.287} C_VEL
LIN {X 0,Y 426.824,Z 683.709,A -85,B 0,C 180,E1 15901.911,E2 15901.911} C_VEL
LIN {X 0,Y 429.872,Z 669.121,A -85,B 0,C 180,E1 15899.765,E2 15899.765} C_VEL
LIN {X 0,Y 433.069,Z 653.017,A -85,B 0,C 180,E1 15897.771,E2 15897.771} C_VEL
LIN {X 0,Y 436.578,Z 634.864,A -85,B 0,C 180,E1 15895.869,E2 15895.869} C_VEL
LIN {X 0,Y 439.873,Z 616.589,A -85,B 0,C 180,E1 15894.256,E2 15894.256} C_VEL
LIN {X 0,Y 442.963,Z 597.265,A -85,B 0,C 180,E1 15892.858,E2 15892.858} C_VEL
LIN {X 0,Y 445.792,Z 577.297,A -85,B 0,C 180,E1 15891.674,E2 15891.674} C_VEL
LIN {X 0,Y 448.089,Z 558.096,A -85,B 0,C 180,E1 15890.759,E2 15890.759} C_VEL
LIN {X 0,Y 450.061,Z 536.68,A -85,B 0,C 180,E1 15889.979,E2 15889.979} C_VEL
LIN {X 0,Y 451.552,Z 514.972,A -85,B 0,C 180,E1 15889.418,E2 15889.418} C_VEL
LIN {X 0,Y 457.579,Z 302.492,A -85,B 0,C 180,E1 15885.769,E2 15885.769} C_VEL
LIN {X 0,Y 459.218,Z 244.36,A -85,B 0,C 180,E1 15884.733,E2 15884.733} C_VEL
LIN {X 0,Y 455.462,Z 219.182,A -85,B 0,C 180,E1 15883.641,E2 15883.641} C_VEL
LIN {X 0,Y 443.911,Z 201.093,A -85,B 0,C 180,E1 15881.441,E2 15881.441} C_VEL
LIN {X 0,Y 436.855,Z 186.443,A -85,B 0,C 180,E1 15878.67,E2 15878.67} C_VEL
LIN {X 0,Y 431.954,Z 177.055,A -85,B 0,C 180,E1 15876.67,E2 15876.67} C_VEL
LIN {X 0,Y 427.849,Z 169.29,A -85,B 0,C 180,E1 15874.891,E2 15874.891} C_VEL
LIN {X 0,Y 425.185,Z 164.523,A -85,B 0,C 180,E1 15873.709,E2 15873.709} C_VEL
LIN {X 0,Y 422.573,Z 159.777,A -85,B 0,C 180,E1 15872.487,E2 15872.487} C_VEL
LIN {X 0,Y 420.571,Z 156.305,A -85,B 0,C 180,E1 15871.536,E2 15871.536} C_VEL
LIN {X 0,Y 419.748,Z 154.818,A -85,B 0,C 180,E1 15871.125,E2 15871.125} C_VEL
LIN {X 0,Y 417.731,Z 151.737,A -85,B 0,C 180,E1 15870.175,E2 15870.175} C_VEL
LIN {X 0,Y 417.336,Z 150.225,A -85,B 0,C 180,E1 15869.731,E2 15869.731} C_VEL
LIN {X 0,Y 417.318,Z 150.012,A -85,B 0,C 180,E1 15866.005,E2 15866.005} C_VEL
LIN {X 0,Y 417.339,Z 150.064,A -85,B 0,C 180,E1 15862.243,E2 15862.243} C_VEL
LIN {X 0,Y 417.349,Z 150.005,A -85,B 0,C 180,E1 15858.435,E2 15858.435} C_VEL
LIN {X 0,Y 417.371,Z 150.045,A -85,B 0,C 180,E1 15854.569,E2 15854.569} C_VEL
LIN {X 0,Y 417.369,Z 150.045,A -85,B 0,C 180,E1 15850.77,E2 15850.77} C_VEL
LIN {X 0,Y 417.375,Z 150.045,A -85,B 0,C 180,E1 15846.88,E2 15846.88} C_VEL
LIN {X 0,Y 417.363,Z 150.048,A -85,B 0,C 180,E1 15843.021,E2 15843.021} C_VEL
LIN {X 0,Y 417.351,Z 150.052,A -85,B 0,C 180,E1 15839.314,E2 15839.314} C_VEL
LIN {X 0,Y 417.348,Z 150.057,A -85,B 0,C 180,E1 15835.466,E2 15835.466} C_VEL
LIN {X 0,Y 417.349,Z 150.059,A -85,B 0,C 180,E1 15831.597,E2 15831.597} C_VEL
LIN {X 0,Y 417.352,Z 150.059,A -85,B 0,C 180,E1 15827.689,E2 15827.689} C_VEL
LIN {X 0,Y 417.348,Z 150.005,A -85,B 0,C 180,E1 15823.722,E2 15823.722} C_VEL
LIN {X 0,Y 417.355,Z 150.02,A -85,B 0,C 180,E1 15819.899,E2 15819.899} C_VEL
LIN {X 0,Y 417.367,Z 150.042,A -85,B 0,C 180,E1 15816.118,E2 15816.118} C_VEL
LIN {X 0,Y 417.4,Z 150.187,A -85,B 0,C 180,E1 15812.618,E2 15812.618} C_VEL
LIN {X 0,Y 417.752,Z 151.65,A -85,B 0,C 180,E1 15812.179,E2 15812.179} C_VEL
LIN {X 0,Y 419.763,Z 154.8,A -85,B 0,C 180,E1 15811.239,E2 15811.239} C_VEL
LIN {X 0,Y 420.66,Z 156.155,A -85,B 0,C 180,E1 15810.84,E2 15810.84} C_VEL
LIN {X 0,Y 422.62,Z 159.785,A -85,B 0,C 180,E1 15809.897,E2 15809.897} C_VEL
LIN {X 0,Y 423.626,Z 161.232,A -85,B 0,C 180,E1 15809.481,E2 15809.481} C_VEL
LIN {X 0,Y 426.004,Z 165.31,A -85,B 0,C 180,E1 15808.44,E2 15808.44} C_VEL
LIN {X 0,Y 429.431,Z 171.465,A -85,B 0,C 180,E1 15807.027,E2 15807.027} C_VEL
LIN {X 0,Y 440.867,Z 186.456,A -85,B 0,C 180,E1 15804.588,E2 15804.588} C_VEL
LIN {X 0,Y 453.103,Z 203.697,A -85,B 0,C 180,E1 15802.22,E2 15802.22} C_VEL
LIN {X 0,Y 463.594,Z 219.964,A -85,B 0,C 180,E1 15800.336,E2 15800.336} C_VEL
LIN {X 0,Y 455.934,Z 434.569,A -85,B 0,C 180,E1 15796.375,E2 15796.375} C_VEL
LIN {X 0,Y 453.111,Z 512.24,A -85,B 0,C 180,E1 15794.919,E2 15794.919} C_VEL
LIN {X 0,Y 451.347,Z 535.371,A -85,B 0,C 180,E1 15794.284,E2 15794.284} C_VEL
LIN {X 0,Y 449.127,Z 558.576,A -85,B 0,C 180,E1 15793.419,E2 15793.419} C_VEL
LIN {X 0,Y 446.801,Z 578.381,A -85,B 0,C 180,E1 15792.473,E2 15792.473} C_VEL
LIN {X 0,Y 443.879,Z 600.2,A -85,B 0,C 180,E1 15791.206,E2 15791.206} C_VEL
LIN {X 0,Y 440.804,Z 620.702,A -85,B 0,C 180,E1 15789.764,E2 15789.764} C_VEL
LIN {X 0,Y 437.494,Z 641.328,A -85,B 0,C 180,E1 15788.042,E2 15788.042} C_VEL
LIN {X 0,Y 434.216,Z 661.182,A -85,B 0,C 180,E1 15786.119,E2 15786.119} C_VEL
LIN {X 0,Y 431.121,Z 678.797,A -85,B 0,C 180,E1 15784.111,E2 15784.111} C_VEL
LIN {X 0,Y 428.135,Z 696.022,A -85,B 0,C 180,E1 15781.856,E2 15781.856} C_VEL
LIN {X 0,Y 425.488,Z 711.029,A -85,B 0,C 180,E1 15779.569,E2 15779.569} C_VEL
LIN {X 0,Y 423.003,Z 725.723,A -85,B 0,C 180,E1 15776.986,E2 15776.986} C_VEL
LIN {X 0,Y 420.974,Z 738.267,A -85,B 0,C 180,E1 15774.41,E2 15774.41} C_VEL
LIN {X 0,Y 419.141,Z 750.776,A -85,B 0,C 180,E1 15771.406,E2 15771.406} C_VEL
LIN {X 0,Y 417.912,Z 760.446,A -85,B 0,C 180,E1 15768.661,E2 15768.661} C_VEL
LIN {X 0,Y 416.989,Z 768.991,A -85,B 0,C 180,E1 15765.72,E2 15765.72} C_VEL
LIN {X 0,Y 416.424,Z 775.6,A -85,B 0,C 180,E1 15762.884,E2 15762.884} C_VEL
LIN {X 0,Y 416.078,Z 781.43,A -85,B 0,C 180,E1 15759.684,E2 15759.684} C_VEL
LIN {X 0,Y 415.961,Z 785.119,A -85,B 0,C 180,E1 15756.903,E2 15756.903} C_VEL
LIN {X 0,Y 415.913,Z 787.848,A -85,B 0,C 180,E1 15753.721,E2 15753.721} C_VEL
LIN {X 0,Y 415.91,Z 788.848,A -85,B 0,C 180,E1 15750.964,E2 15750.964} C_VEL
LIN {X 0,Y 415.905,Z 788.658,A -85,B 0,C 180,E1 15747.933,E2 15747.933} C_VEL
LIN {X 0,Y 415.92,Z 786.84,A -85,B 0,C 180,E1 15744.897,E2 15744.897} C_VEL
LIN {X 0,Y 416.003,Z 783.839,A -85,B 0,C 180,E1 15741.985,E2 15741.985} C_VEL
LIN {X 0,Y 416.204,Z 779.082,A -85,B 0,C 180,E1 15738.92,E2 15738.92} C_VEL
LIN {X 0,Y 416.626,Z 773.134,A -85,B 0,C 180,E1 15735.973,E2 15735.973} C_VEL
LIN {X 0,Y 417.37,Z 765.253,A -85,B 0,C 180,E1 15732.91,E2 15732.91} C_VEL
LIN {X 0,Y 418.454,Z 756.055,A -85,B 0,C 180,E1 15730.021,E2 15730.021} C_VEL
LIN {X 0,Y 419.963,Z 744.944,A -85,B 0,C 180,E1 15727.128,E2 15727.128} C_VEL
LIN {X 0,Y 421.936,Z 732.278,A -85,B 0,C 180,E1 15724.301,E2 15724.301} C_VEL
LIN {X 0,Y 424.186,Z 718.649,A -85,B 0,C 180,E1 15721.721,E2 15721.721} C_VEL
LIN {X 0,Y 426.977,Z 702.539,A -85,B 0,C 180,E1 15719.098,E2 15719.098} C_VEL
LIN {X 0,Y 429.792,Z 686.544,A -85,B 0,C 180,E1 15716.86,E2 15716.86} C_VEL
LIN {X 0,Y 432.972,Z 668.185,A -85,B 0,C 180,E1 15714.65,E2 15714.65} C_VEL
LIN {X 0,Y 436.192,Z 649.352,A -85,B 0,C 180,E1 15712.693,E2 15712.693} C_VEL
LIN {X 0,Y 439.435,Z 629.417,A -85,B 0,C 180,E1 15710.932,E2 15710.932} C_VEL
LIN {X 0,Y 442.731,Z 608.042,A -85,B 0,C 180,E1 15709.315,E2 15709.315} C_VEL
LIN {X 0,Y 445.574,Z 587.699,A -85,B 0,C 180,E1 15708.034,E2 15708.034} C_VEL
LIN {X 0,Y 448.356,Z 565.313,A -85,B 0,C 180,E1 15706.883,E2 15706.883} C_VEL
LIN {X 0,Y 450.605,Z 544.082,A -85,B 0,C 180,E1 15706.012,E2 15706.012} C_VEL
LIN {X 0,Y 452.49,Z 521.235,A -85,B 0,C 180,E1 15705.309,E2 15705.309} C_VEL
LIN {X 0,Y 453.791,Z 497.726,A -85,B 0,C 180,E1 15704.787,E2 15704.787} C_VEL
LIN {X 0,Y 461.177,Z 286.52,A -85,B 0,C 180,E1 15700.893,E2 15700.893} C_VEL
LIN {X 0,Y 463.49,Z 219.622,A -85,B 0,C 180,E1 15699.643,E2 15699.643} C_VEL
LIN {X 0,Y 451.383,Z 201.303,A -85,B 0,C 180,E1 15697.468,E2 15697.468} C_VEL
LIN {X 0,Y 440.024,Z 185.298,A -85,B 0,C 180,E1 15695.251,E2 15695.251} C_VEL
LIN {X 0,Y 431.4,Z 174.18,A -85,B 0,C 180,E1 15693.438,E2 15693.438} C_VEL
LIN {X 0,Y 428.757,Z 170.202,A -85,B 0,C 180,E1 15692.753,E2 15692.753} C_VEL
LIN {X 0,Y 425.606,Z 164.836,A -85,B 0,C 180,E1 15691.435,E2 15691.435} C_VEL
LIN {X 0,Y 422.917,Z 160.114,A -85,B 0,C 180,E1 15690.236,E2 15690.236} C_VEL
LIN {X 0,Y 420.842,Z 156.699,A -85,B 0,C 180,E1 15689.303,E2 15689.303} C_VEL
LIN {X 0,Y 420.058,Z 155.079,A -85,B 0,C 180,E1 15688.894,E2 15688.894} C_VEL
LIN {X 0,Y 417.932,Z 152.132,A -85,B 0,C 180,E1 15687.963,E2 15687.963} C_VEL
LIN {X 0,Y 417.417,Z 150.298,A -85,B 0,C 180,E1 15687.476,E2 15687.476} C_VEL
LIN {X 0,Y 417.38,Z 150.042,A -85,B 0,C 180,E1 15685.088,E2 15685.088} C_VEL
LIN {X 0,Y 417.376,Z 150.001,A -85,B 0,C 180,E1 15681.206,E2 15681.206} C_VEL
LIN {X 0,Y 417.378,Z 150.03,A -85,B 0,C 180,E1 15677.424,E2 15677.424} C_VEL
LIN {X 0,Y 417.375,Z 150.019,A -85,B 0,C 180,E1 15673.578,E2 15673.578} C_VEL
LIN {X 0,Y 417.37,Z 150.045,A -85,B 0,C 180,E1 15669.654,E2 15669.654} C_VEL
LIN {X 0,Y 417.355,Z 150.053,A -85,B 0,C 180,E1 15665.913,E2 15665.913} C_VEL
LIN {X 0,Y 417.348,Z 150.06,A -85,B 0,C 180,E1 15662.059,E2 15662.059} C_VEL
LIN {X 0,Y 417.343,Z 150.062,A -85,B 0,C 180,E1 15658.215,E2 15658.215} C_VEL
LIN {X 0,Y 417.341,Z 150.063,A -85,B 0,C 180,E1 15654.363,E2 15654.363} C_VEL
LIN {X 0,Y 417.345,Z 150.061,A -85,B 0,C 180,E1 15650.624,E2 15650.624} C_VEL
LIN {X 0,Y 417.355,Z 150.056,A -85,B 0,C 180,E1 15646.844,E2 15646.844} C_VEL
LIN {X 0,Y 417.372,Z 150.044,A -85,B 0,C 180,E1 15643.15,E2 15643.15} C_VEL
LIN {X 0,Y 417.371,Z 150.016,A -85,B 0,C 180,E1 15639.234,E2 15639.234} C_VEL
LIN {X 0,Y 417.352,Z 150.011,A -85,B 0,C 180,E1 15635.514,E2 15635.514} C_VEL
LIN {X 0,Y 417.342,Z 150.063,A -85,B 0,C 180,E1 15631.682,E2 15631.682} C_VEL
LIN {X 0,Y 417.353,Z 150.297,A -85,B 0,C 180,E1 15630.112,E2 15630.112} C_VEL
LIN {X 0,Y 418.866,Z 153.78,A -85,B 0,C 180,E1 15629.121,E2 15629.121} C_VEL
LIN {X 0,Y 420.424,Z 155.823,A -85,B 0,C 180,E1 15628.452,E2 15628.452} C_VEL
LIN {X 0,Y 422.334,Z 159.486,A -85,B 0,C 180,E1 15627.492,E2 15627.492} C_VEL
LIN {X 0,Y 423.28,Z 160.854,A -85,B 0,C 180,E1 15627.091,E2 15627.091} C_VEL
LIN {X 0,Y 425.292,Z 164.651,A -85,B 0,C 180,E1 15626.138,E2 15626.138} C_VEL
LIN {X 0,Y 430.879,Z 174.688,A -85,B 0,C 180,E1 15623.72,E2 15623.72} C_VEL
LIN {X 0,Y 437.971,Z 188.718,A -85,B 0,C 180,E1 15620.774,E2 15620.774} C_VEL
LIN {X 0,Y 444.24,Z 201.696,A -85,B 0,C 180,E1 15618.376,E2 15618.376} C_VEL
LIN {X 0,Y 455.591,Z 219.439,A -85,B 0,C 180,E1 15616.236,E2 15616.236} C_VEL
LIN {X 0,Y 459.287,Z 246.129,A -85,B 0,C 180,E1 15615.12,E2 15615.12} C_VEL
LIN {X 0,Y 452.793,Z 473.683,A -85,B 0,C 180,E1 15611.212,E2 15611.212} C_VEL
LIN {X 0,Y 451.397,Z 517.936,A -85,B 0,C 180,E1 15610.429,E2 15610.429} C_VEL
LIN {X 0,Y 450.465,Z 531.785,A -85,B 0,C 180,E1 15610.079,E2 15610.079} C_VEL
LIN {X 0,Y 448.969,Z 539.331,A -85,B 0,C 180,E1 15609.951,E2 15609.951} C_VEL
LIN {X 0,Y 443.012,Z 557.508,A -85,B 0,C 180,E1 15609.775,E2 15609.775} C_VEL
LIN {X 0,Y 441.336,Z 564.695,A -85,B 0,C 180,E1 15609.553,E2 15609.553} C_VEL
LIN {X 0,Y 441.198,Z 565.715,A -85,B 0,C 180,E1 15609.509,E2 15609.509} C_VEL
LIN {X 0,Y 438.418,Z 586.326,A -85,B 0,C 180,E1 15608.422,E2 15608.422} C_VEL
LIN {X 0,Y 435.4,Z 605.801,A -85,B 0,C 180,E1 15607.153,E2 15607.153} C_VEL
LIN {X 0,Y 432.074,Z 624.353,A -85,B 0,C 180,E1 15605.671,E2 15605.671} C_VEL
LIN {X 0,Y 428.458,Z 642.934,A -85,B 0,C 180,E1 15603.898,E2 15603.898} C_VEL
LIN {X 0,Y 424.966,Z 660.041,A -85,B 0,C 180,E1 15601.963,E2 15601.963} C_VEL
LIN {X 0,Y 421.495,Z 676.06,A -85,B 0,C 180,E1 15599.799,E2 15599.799} C_VEL
LIN {X 0,Y 418.336,Z 690.729,A -85,B 0,C 180,E1 15597.469,E2 15597.469} C_VEL
LIN {X 0,Y 415.596,Z 703.735,A -85,B 0,C 180,E1 15595.05,E2 15595.05} C_VEL
LIN {X 0,Y 413.121,Z 715.993,A -85,B 0,C 180,E1 15592.332,E2 15592.332} C_VEL
LIN {X 0,Y 411.081,Z 727.455,A -85,B 0,C 180,E1 15589.313,E2 15589.313} C_VEL
LIN {X 0,Y 409.666,Z 736.949,A -85,B 0,C 180,E1 15586.3,E2 15586.3} C_VEL
LIN {X 0,Y 408.767,Z 744.612,A -85,B 0,C 180,E1 15583.292,E2 15583.292} C_VEL
LIN {X 0,Y 408.252,Z 750.6,A -85,B 0,C 180,E1 15580.299,E2 15580.299} C_VEL
LIN {X 0,Y 408.024,Z 755.091,A -85,B 0,C 180,E1 15577.321,E2 15577.321} C_VEL
LIN {X 0,Y 407.939,Z 757.954,A -85,B 0,C 180,E1 15574.357,E2 15574.357} C_VEL
LIN {X 0,Y 407.917,Z 759.438,A -85,B 0,C 180,E1 15571.264,E2 15571.264} C_VEL
LIN {X 0,Y 407.918,Z 759.409,A -85,B 0,C 180,E1 15568.455,E2 15568.455} C_VEL
LIN {X 0,Y 407.94,Z 757.914,A -85,B 0,C 180,E1 15565.502,E2 15565.502} C_VEL
LIN {X 0,Y 408.022,Z 755.033,A -85,B 0,C 180,E1 15562.538,E2 15562.538} C_VEL
LIN {X 0,Y 408.259,Z 750.502,A -85,B 0,C 180,E1 15559.559,E2 15559.559} C_VEL
LIN {X 0,Y 408.81,Z 744.141,A -85,B 0,C 180,E1 15556.421,E2 15556.421} C_VEL
LIN {X 0,Y 409.75,Z 736.41,A -85,B 0,C 180,E1 15553.412,E2 15553.412} C_VEL
LIN {X 0,Y 411.198,Z 726.749,A -85,B 0,C 180,E1 15550.394,E2 15550.394} C_VEL
LIN {X 0,Y 413.164,Z 715.739,A -85,B 0,C 180,E1 15547.521,E2 15547.521} C_VEL
LIN {X 0,Y 415.653,Z 703.439,A -85,B 0,C 180,E1 15544.801,E2 15544.801} C_VEL
LIN {X 0,Y 418.41,Z 690.395,A -85,B 0,C 180,E1 15542.382,E2 15542.382} C_VEL
LIN {X 0,Y 421.691,Z 675.16,A -85,B 0,C 180,E1 15539.981,E2 15539.981} C_VEL
LIN {X 0,Y 425.126,Z 659.281,A -85,B 0,C 180,E1 15537.854,E2 15537.854} C_VEL
LIN {X 0,Y 428.703,Z 641.796,A -85,B 0,C 180,E1 15535.89,E2 15535.89} C_VEL
LIN {X 0,Y 432.211,Z 623.668,A -85,B 0,C 180,E1 15534.178,E2 15534.178} C_VEL
LIN {X 0,Y 435.545,Z 604.997,A -85,B 0,C 180,E1 15532.697,E2 15532.697} C_VEL
LIN {X 0,Y 438.52,Z 585.72,A -85,B 0,C 180,E1 15531.45,E2 15531.45} C_VEL
LIN {X 0,Y 441.366,Z 564.395,A -85,B 0,C 180,E1 15530.34,E2 15530.34} C_VEL
LIN {X 0,Y 443.603,Z 543.864,A -85,B 0,C 180,E1 15529.509,E2 15529.509} C_VEL
LIN {X 0,Y 445.263,Z 522.65,A -85,B 0,C 180,E1 15528.89,E2 15528.89} C_VEL
LIN {X 0,Y 446.455,Z 495.496,A -85,B 0,C 180,E1 15528.356,E2 15528.356} C_VEL
LIN {X 0,Y 453.174,Z 269.336,A -85,B 0,C 180,E1 15524.444,E2 15524.444} C_VEL
LIN {X 0,Y 453.801,Z 245.867,A -85,B 0,C 180,E1 15524.006,E2 15524.006} C_VEL
LIN {X 0,Y 450.581,Z 223.705,A -85,B 0,C 180,E1 15523.028,E2 15523.028} C_VEL
LIN {X 0,Y 439.362,Z 206.116,A -85,B 0,C 180,E1 15520.843,E2 15520.843} C_VEL
LIN {X 0,Y 435.09,Z 199.509,A -85,B 0,C 180,E1 15519.878,E2 15519.878} C_VEL
LIN {X 0,Y 429.208,Z 187.494,A -85,B 0,C 180,E1 15517.446,E2 15517.446} C_VEL
LIN {X 0,Y 422.989,Z 175.53,A -85,B 0,C 180,E1 15514.728,E2 15514.728} C_VEL
LIN {X 0,Y 419.949,Z 170.2,A -85,B 0,C 180,E1 15513.366,E2 15513.366} C_VEL
LIN {X 0,Y 417.69,Z 165.937,A -85,B 0,C 180,E1 15512.264,E2 15512.264} C_VEL
LIN {X 0,Y 415.501,Z 161.846,A -85,B 0,C 180,E1 15511.157,E2 15511.157} C_VEL
LIN {X 0,Y 412.898,Z 157.796,A -85,B 0,C 180,E1 15509.9,E2 15509.9} C_VEL
LIN {X 0,Y 411.928,Z 155.942,A -85,B 0,C 180,E1 15509.361,E2 15509.361} C_VEL
LIN {X 0,Y 409.766,Z 152.657,A -85,B 0,C 180,E1 15508.254,E2 15508.254} C_VEL
LIN {X 0,Y 409.385,Z 151.113,A -85,B 0,C 180,E1 15507.693,E2 15507.693} C_VEL
LIN {X 0,Y 409.378,Z 151.014,A -85,B 0,C 180,E1 15503.766,E2 15503.766} C_VEL
LIN {X 0,Y 409.382,Z 150.995,A -85,B 0,C 180,E1 15499.901,E2 15499.901} C_VEL
LIN {X 0,Y 409.393,Z 151.054,A -85,B 0,C 180,E1 15496.021,E2 15496.021} C_VEL
LIN {X 0,Y 409.409,Z 151.05,A -85,B 0,C 180,E1 15492.267,E2 15492.267} C_VEL
LIN {X 0,Y 409.424,Z 151.042,A -85,B 0,C 180,E1 15488.426,E2 15488.426} C_VEL
LIN {X 0,Y 409.434,Z 151.036,A -85,B 0,C 180,E1 15484.623,E2 15484.623} C_VEL
LIN {X 0,Y 409.446,Z 151.031,A -85,B 0,C 180,E1 15480.7,E2 15480.7} C_VEL
LIN {X 0,Y 409.437,Z 151.031,A -85,B 0,C 180,E1 15476.78,E2 15476.78} C_VEL
LIN {X 0,Y 409.447,Z 151.03,A -85,B 0,C 180,E1 15472.846,E2 15472.846} C_VEL
LIN {X 0,Y 409.438,Z 151.033,A -85,B 0,C 180,E1 15468.877,E2 15468.877} C_VEL
LIN {X 0,Y 409.439,Z 150.982,A -85,B 0,C 180,E1 15464.998,E2 15464.998} C_VEL
LIN {X 0,Y 409.439,Z 151.041,A -85,B 0,C 180,E1 15461.047,E2 15461.047} C_VEL
LIN {X 0,Y 409.436,Z 150.999,A -85,B 0,C 180,E1 15457.152,E2 15457.152} C_VEL
LIN {X 0,Y 409.487,Z 151.345,A -85,B 0,C 180,E1 15454.471,E2 15454.471} C_VEL
LIN {X 0,Y 411.022,Z 154.888,A -85,B 0,C 180,E1 15453.41,E2 15453.41} C_VEL
LIN {X 0,Y 412.805,Z 157.168,A -85,B 0,C 180,E1 15452.6,E2 15452.6} C_VEL
LIN {X 0,Y 414.622,Z 160.636,A -85,B 0,C 180,E1 15451.637,E2 15451.637} C_VEL
LIN {X 0,Y 415.854,Z 162.306,A -85,B 0,C 180,E1 15451.101,E2 15451.101} C_VEL
LIN {X 0,Y 418.114,Z 166.34,A -85,B 0,C 180,E1 15450.014,E2 15450.014} C_VEL
LIN {X 0,Y 421.743,Z 172.428,A -85,B 0,C 180,E1 15448.483,E2 15448.483} C_VEL
LIN {X 0,Y 431.354,Z 184.94,A -85,B 0,C 180,E1 15446.279,E2 15446.279} C_VEL
LIN {X 0,Y 441.196,Z 198.285,A -85,B 0,C 180,E1 15444.219,E2 15444.219} C_VEL
LIN {X 0,Y 452.2,Z 214.342,A -85,B 0,C 180,E1 15442.091,E2 15442.091} C_VEL
LIN {X 0,Y 458.091,Z 223.797,A -85,B 0,C 180,E1 15441.009,E2 15441.009} C_VEL
LIN {X 0,Y 449.983,Z 439.918,A -85,B 0,C 180,E1 15436.982,E2 15436.982} C_VEL
LIN {X 0,Y 447.195,Z 512.433,A -85,B 0,C 180,E1 15435.606,E2 15435.606} C_VEL
LIN {X 0,Y 445.336,Z 535.599,A -85,B 0,C 180,E1 15434.963,E2 15434.963} C_VEL
LIN {X 0,Y 443.003,Z 558.796,A -85,B 0,C 180,E1 15434.088,E2 15434.088} C_VEL
LIN {X 0,Y 440.558,Z 578.591,A -85,B 0,C 180,E1 15433.132,E2 15433.132} C_VEL
LIN {X 0,Y 437.343,Z 601.241,A -85,B 0,C 180,E1 15431.791,E2 15431.791} C_VEL
LIN {X 0,Y 434.117,Z 621.627,A -85,B 0,C 180,E1 15430.329,E2 15430.329} C_VEL
LIN {X 0,Y 430.614,Z 641.989,A -85,B 0,C 180,E1 15428.586,E2 15428.586} C_VEL
LIN {X 0,Y 427.153,Z 661.424,A -85,B 0,C 180,E1 15426.646,E2 15426.646} C_VEL
LIN {X 0,Y 423.625,Z 680.415,A -85,B 0,C 180,E1 15424.425,E2 15424.425} C_VEL
LIN {X 0,Y 420.378,Z 698.022,A -85,B 0,C 180,E1 15422.031,E2 15422.031} C_VEL
LIN {X 0,Y 417.663,Z 712.857,A -85,B 0,C 180,E1 15419.705,E2 15419.705} C_VEL
LIN {X 0,Y 415.101,Z 727.238,A -85,B 0,C 180,E1 15417.08,E2 15417.08} C_VEL
LIN {X 0,Y 413.028,Z 739.687,A -85,B 0,C 180,E1 15414.453,E2 15414.453} C_VEL
LIN {X 0,Y 411.22,Z 751.349,A -85,B 0,C 180,E1 15411.539,E2 15411.539} C_VEL
LIN {X 0,Y 409.907,Z 761.298,A -85,B 0,C 180,E1 15408.635,E2 15408.635} C_VEL
LIN {X 0,Y 408.957,Z 769.849,A -85,B 0,C 180,E1 15405.574,E2 15405.574} C_VEL
LIN {X 0,Y 408.394,Z 776.732,A -85,B 0,C 180,E1 15402.585,E2 15402.585} C_VEL
LIN {X 0,Y 408.079,Z 781.843,A -85,B 0,C 180,E1 15399.591,E2 15399.591} C_VEL
LIN {X 0,Y 407.959,Z 785.438,A -85,B 0,C 180,E1 15396.756,E2 15396.756} C_VEL
LIN {X 0,Y 407.91,Z 787.983,A -85,B 0,C 180,E1 15393.513,E2 15393.513} C_VEL
LIN {X 0,Y 407.906,Z 788.871,A -85,B 0,C 180,E1 15390.843,E2 15390.843} C_VEL
LIN {X 0,Y 407.906,Z 788.595,A -85,B 0,C 180,E1 15387.752,E2 15387.752} C_VEL
LIN {X 0,Y 407.921,Z 786.84,A -85,B 0,C 180,E1 15384.797,E2 15384.797} C_VEL
LIN {X 0,Y 408.009,Z 783.84,A -85,B 0,C 180,E1 15381.829,E2 15381.829} C_VEL
LIN {X 0,Y 408.233,Z 779.082,A -85,B 0,C 180,E1 15378.701,E2 15378.701} C_VEL
LIN {X 0,Y 408.63,Z 773.606,A -85,B 0,C 180,E1 15375.982,E2 15375.982} C_VEL
LIN {X 0,Y 409.435,Z 765.25,A -85,B 0,C 180,E1 15372.714,E2 15372.714} C_VEL
LIN {X 0,Y 410.576,Z 756.07,A -85,B 0,C 180,E1 15369.77,E2 15369.77} C_VEL
LIN {X 0,Y 412.153,Z 745.096,A -85,B 0,C 180,E1 15366.842,E2 15366.842} C_VEL
LIN {X 0,Y 414.127,Z 733.068,A -85,B 0,C 180,E1 15364.088,E2 15364.088} C_VEL
LIN {X 0,Y 416.462,Z 719.501,A -85,B 0,C 180,E1 15361.461,E2 15361.461} C_VEL
LIN {X 0,Y 419.317,Z 703.891,A -85,B 0,C 180,E1 15358.841,E2 15358.841} C_VEL
LIN {X 0,Y 422.292,Z 687.69,A -85,B 0,C 180,E1 15356.519,E2 15356.519} C_VEL
LIN {X 0,Y 425.9,Z 667.97,A -85,B 0,C 180,E1 15354.089,E2 15354.089} C_VEL
LIN {X 0,Y 429.484,Z 648.594,A -85,B 0,C 180,E1 15352.033,E2 15352.033} C_VEL
LIN {X 0,Y 432.95,Z 628.514,A -85,B 0,C 180,E1 15350.231,E2 15350.231} C_VEL
LIN {X 0,Y 436.538,Z 606.377,A -85,B 0,C 180,E1 15348.554,E2 15348.554} C_VEL
LIN {X 0,Y 439.633,Z 585.501,A -85,B 0,C 180,E1 15347.243,E2 15347.243} C_VEL
LIN {X 0,Y 442.31,Z 564.586,A -85,B 0,C 180,E1 15346.175,E2 15346.175} C_VEL
LIN {X 0,Y 444.634,Z 543.571,A -85,B 0,C 180,E1 15345.31,E2 15345.31} C_VEL
LIN {X 0,Y 446.581,Z 520.817,A -85,B 0,C 180,E1 15344.61,E2 15344.61} C_VEL
LIN {X 0,Y 447.933,Z 497.072,A -85,B 0,C 180,E1 15344.082,E2 15344.082} C_VEL
LIN {X 0,Y 455.699,Z 286.312,A -85,B 0,C 180,E1 15340.156,E2 15340.156} C_VEL
LIN {X 0,Y 457.948,Z 223.306,A -85,B 0,C 180,E1 15338.962,E2 15338.962} C_VEL
LIN {X 0,Y 445.691,Z 204.675,A -85,B 0,C 180,E1 15336.677,E2 15336.677} C_VEL
LIN {X 0,Y 433.158,Z 187.175,A -85,B 0,C 180,E1 15334.119,E2 15334.119} C_VEL
LIN {X 0,Y 424.267,Z 175.811,A -85,B 0,C 180,E1 15332.142,E2 15332.142} C_VEL
LIN {X 0,Y 421.099,Z 171.415,A -85,B 0,C 180,E1 15331.332,E2 15331.332} C_VEL
LIN {X 0,Y 417.729,Z 165.873,A -85,B 0,C 180,E1 15329.858,E2 15329.858} C_VEL
LIN {X 0,Y 415.224,Z 161.299,A -85,B 0,C 180,E1 15328.632,E2 15328.632} C_VEL
LIN {X 0,Y 412.966,Z 157.668,A -85,B 0,C 180,E1 15327.545,E2 15327.545} C_VEL
LIN {X 0,Y 412.097,Z 156.021,A -85,B 0,C 180,E1 15327.075,E2 15327.075} C_VEL
LIN {X 0,Y 409.944,Z 153.018,A -85,B 0,C 180,E1 15326.041,E2 15326.041} C_VEL
LIN {X 0,Y 409.476,Z 151.281,A -85,B 0,C 180,E1 15325.529,E2 15325.529} C_VEL
LIN {X 0,Y 409.436,Z 150.987,A -85,B 0,C 180,E1 15321.638,E2 15321.638} C_VEL
LIN {X 0,Y 409.43,Z 151.028,A -85,B 0,C 180,E1 15317.753,E2 15317.753} C_VEL
LIN {X 0,Y 409.421,Z 151,A -85,B 0,C 180,E1 15313.847,E2 15313.847} C_VEL
LIN {X 0,Y 409.416,Z 151.033,A -85,B 0,C 180,E1 15309.985,E2 15309.985} C_VEL
LIN {X 0,Y 409.409,Z 151.038,A -85,B 0,C 180,E1 15306.169,E2 15306.169} C_VEL
LIN {X 0,Y 409.406,Z 151.045,A -85,B 0,C 180,E1 15302.239,E2 15302.239} C_VEL
LIN {X 0,Y 409.404,Z 151.05,A -85,B 0,C 180,E1 15298.32,E2 15298.32} C_VEL
LIN {X 0,Y 409.402,Z 151.052,A -85,B 0,C 180,E1 15294.394,E2 15294.394} C_VEL
LIN {X 0,Y 409.405,Z 151.05,A -85,B 0,C 180,E1 15290.582,E2 15290.582} C_VEL
LIN {X 0,Y 409.408,Z 151.044,A -85,B 0,C 180,E1 15286.728,E2 15286.728} C_VEL
LIN {X 0,Y 409.418,Z 151.025,A -85,B 0,C 180,E1 15282.959,E2 15282.959} C_VEL
LIN {X 0,Y 409.426,Z 151.006,A -85,B 0,C 180,E1 15279.112,E2 15279.112} C_VEL
LIN {X 0,Y 409.422,Z 150.993,A -85,B 0,C 180,E1 15275.291,E2 15275.291} C_VEL
LIN {X 0,Y 409.422,Z 151.307,A -85,B 0,C 180,E1 15272.038,E2 15272.038} C_VEL
LIN {X 0,Y 411.068,Z 154.999,A -85,B 0,C 180,E1 15270.891,E2 15270.891} C_VEL
LIN {X 0,Y 412.644,Z 157.033,A -85,B 0,C 180,E1 15270.161,E2 15270.161} C_VEL
LIN {X 0,Y 414.65,Z 160.742,A -85,B 0,C 180,E1 15269.095,E2 15269.095} C_VEL
LIN {X 0,Y 415.601,Z 162.166,A -85,B 0,C 180,E1 15268.654,E2 15268.654} C_VEL
LIN {X 0,Y 417.784,Z 166.047,A -85,B 0,C 180,E1 15267.582,E2 15267.582} C_VEL
LIN {X 0,Y 421.546,Z 173.015,A -85,B 0,C 180,E1 15265.796,E2 15265.796} C_VEL
LIN {X 0,Y 425.96,Z 181.131,A -85,B 0,C 180,E1 15263.847,E2 15263.847} C_VEL
LIN {X 0,Y 432.582,Z 194.26,A -85,B 0,C 180,E1 15261.046,E2 15261.046} C_VEL
LIN {X 0,Y 436.197,Z 201.369,A -85,B 0,C 180,E1 15259.707,E2 15259.707} C_VEL
LIN {X 0,Y 449.122,Z 221.327,A -85,B 0,C 180,E1 15257.147,E2 15257.147} C_VEL
LIN {X 0,Y 450.788,Z 224.536,A -85,B 0,C 180,E1 15256.822,E2 15256.822} C_VEL
LIN {X 0,Y 453.873,Z 247.74,A -85,B 0,C 180,E1 15255.842,E2 15255.842} C_VEL
LIN {X 0,Y 447.019,Z 474.575,A -85,B 0,C 180,E1 15251.91,E2 15251.91} C_VEL
LIN {X 0,Y 445.572,Z 517.934,A -85,B 0,C 180,E1 15251.134,E2 15251.134} C_VEL
LIN {X 0,Y 443.965,Z 539.208,A -85,B 0,C 180,E1 15250.552,E2 15250.552} C_VEL
LIN {X 0,Y 441.813,Z 560.539,A -85,B 0,C 180,E1 15249.74,E2 15249.74} C_VEL
LIN {X 0,Y 441.198,Z 565.715,A -85,B 0,C 180,E1 15249.509,E2 15249.509} C_VEL
LIN {X 0,Y 439.541,Z 573.042,A -85,B 0,C 180,E1 15249.249,E2 15249.249} C_VEL
LIN {X 0,Y 432.331,Z 591.428,A -85,B 0,C 180,E1 15248.735,E2 15248.735} C_VEL
LIN {X 0,Y 430.419,Z 598.365,A -85,B 0,C 180,E1 15248.367,E2 15248.367} C_VEL
LIN {X 0,Y 427.128,Z 617.101,A -85,B 0,C 180,E1 15246.984,E2 15246.984} C_VEL
LIN {X 0,Y 423.496,Z 635.392,A -85,B 0,C 180,E1 15245.339,E2 15245.339} C_VEL
LIN {X 0,Y 419.634,Z 653.578,A -85,B 0,C 180,E1 15243.393,E2 15243.393} C_VEL
LIN {X 0,Y 416.062,Z 669.754,A -85,B 0,C 180,E1 15241.35,E2 15241.35} C_VEL
LIN {X 0,Y 412.681,Z 684.453,A -85,B 0,C 180,E1 15239.142,E2 15239.142} C_VEL
LIN {X 0,Y 409.355,Z 699.164,A -85,B 0,C 180,E1 15236.549,E2 15236.549} C_VEL
LIN {X 0,Y 406.639,Z 711.742,A -85,B 0,C 180,E1 15233.935,E2 15233.935} C_VEL
LIN {X 0,Y 404.364,Z 722.843,A -85,B 0,C 180,E1 15231.162,E2 15231.162} C_VEL
LIN {X 0,Y 402.442,Z 733.597,A -85,B 0,C 180,E1 15227.943,E2 15227.943} C_VEL
LIN {X 0,Y 401.239,Z 741.988,A -85,B 0,C 180,E1 15224.872,E2 15224.872} C_VEL
LIN {X 0,Y 400.506,Z 748.615,A -85,B 0,C 180,E1 15221.812,E2 15221.812} C_VEL
LIN {X 0,Y 400.118,Z 753.861,A -85,B 0,C 180,E1 15218.623,E2 15218.623} C_VEL
LIN {X 0,Y 399.972,Z 757.385,A -85,B 0,C 180,E1 15215.595,E2 15215.595} C_VEL
LIN {X 0,Y 399.924,Z 759.316,A -85,B 0,C 180,E1 15212.579,E2 15212.579} C_VEL
LIN {X 0,Y 399.917,Z 759.853,A -85,B 0,C 180,E1 15209.427,E2 15209.427} C_VEL
LIN {X 0,Y 399.935,Z 758.964,A -85,B 0,C 180,E1 15206.56,E2 15206.56} C_VEL
LIN {X 0,Y 400,Z 756.428,A -85,B 0,C 180,E1 15203.397,E2 15203.397} C_VEL
LIN {X 0,Y 400.206,Z 752.572,A -85,B 0,C 180,E1 15200.364,E2 15200.364} C_VEL
LIN {X 0,Y 400.654,Z 747.05,A -85,B 0,C 180,E1 15197.314,E2 15197.314} C_VEL
LIN {X 0,Y 401.551,Z 739.583,A -85,B 0,C 180,E1 15194.104,E2 15194.104} C_VEL
LIN {X 0,Y 402.936,Z 730.732,A -85,B 0,C 180,E1 15191.031,E2 15191.031} C_VEL
LIN {X 0,Y 404.842,Z 720.438,A -85,B 0,C 180,E1 15188.104,E2 15188.104} C_VEL
LIN {X 0,Y 407.308,Z 708.491,A -85,B 0,C 180,E1 15185.268,E2 15185.268} C_VEL
LIN {X 0,Y 410.127,Z 695.83,A -85,B 0,C 180,E1 15182.721,E2 15182.721} C_VEL
LIN {X 0,Y 413.42,Z 681.258,A -85,B 0,C 180,E1 15180.255,E2 15180.255} C_VEL
LIN {X 0,Y 416.985,Z 665.531,A -85,B 0,C 180,E1 15178.001,E2 15178.001} C_VEL
LIN {X 0,Y 420.699,Z 648.864,A -85,B 0,C 180,E1 15175.969,E2 15175.969} C_VEL
LIN {X 0,Y 424.212,Z 631.898,A -85,B 0,C 180,E1 15174.231,E2 15174.231} C_VEL
LIN {X 0,Y 427.906,Z 612.809,A -85,B 0,C 180,E1 15172.591,E2 15172.591} C_VEL
LIN {X 0,Y 431.212,Z 593.925,A -85,B 0,C 180,E1 15171.242,E2 15171.242} C_VEL
LIN {X 0,Y 434.133,Z 574.173,A -85,B 0,C 180,E1 15170.104,E2 15170.104} C_VEL
LIN {X 0,Y 436.778,Z 552.717,A -85,B 0,C 180,E1 15169.121,E2 15169.121} C_VEL
LIN {X 0,Y 438.842,Z 531.582,A -85,B 0,C 180,E1 15168.399,E2 15168.399} C_VEL
LIN {X 0,Y 440.225,Z 509.825,A -85,B 0,C 180,E1 15167.889,E2 15167.889} C_VEL
LIN {X 0,Y 447.305,Z 285.329,A -85,B 0,C 180,E1 15163.964,E2 15163.964} C_VEL
LIN {X 0,Y 448.48,Z 247.541,A -85,B 0,C 180,E1 15163.268,E2 15163.268} C_VEL
LIN {X 0,Y 445.684,Z 228.1,A -85,B 0,C 180,E1 15162.388,E2 15162.388} C_VEL
LIN {X 0,Y 434.977,Z 211.234,A -85,B 0,C 180,E1 15160.235,E2 15160.235} C_VEL
LIN {X 0,Y 427.129,Z 199.521,A -85,B 0,C 180,E1 15158.512,E2 15158.512} C_VEL
LIN {X 0,Y 420.178,Z 185.684,A -85,B 0,C 180,E1 15155.495,E2 15155.495} C_VEL
LIN {X 0,Y 415.376,Z 176.794,A -85,B 0,C 180,E1 15153.286,E2 15153.286} C_VEL
LIN {X 0,Y 412.499,Z 171.665,A -85,B 0,C 180,E1 15151.898,E2 15151.898} C_VEL
LIN {X 0,Y 409.868,Z 166.965,A -85,B 0,C 180,E1 15150.559,E2 15150.559} C_VEL
LIN {X 0,Y 407.43,Z 162.499,A -85,B 0,C 180,E1 15149.233,E2 15149.233} C_VEL
LIN {X 0,Y 405.038,Z 158.792,A -85,B 0,C 180,E1 15147.971,E2 15147.971} C_VEL
LIN {X 0,Y 404.089,Z 157.035,A -85,B 0,C 180,E1 15147.402,E2 15147.402} C_VEL
LIN {X 0,Y 401.831,Z 153.635,A -85,B 0,C 180,E1 15146.131,E2 15146.131} C_VEL
LIN {X 0,Y 401.448,Z 152.071,A -85,B 0,C 180,E1 15145.524,E2 15145.524} C_VEL
LIN {X 0,Y 401.442,Z 152.022,A -85,B 0,C 180,E1 15141.631,E2 15141.631} C_VEL
LIN {X 0,Y 401.444,Z 151.994,A -85,B 0,C 180,E1 15137.69,E2 15137.69} C_VEL
LIN {X 0,Y 401.452,Z 152.028,A -85,B 0,C 180,E1 15133.687,E2 15133.687} C_VEL
LIN {X 0,Y 401.456,Z 152.035,A -85,B 0,C 180,E1 15129.751,E2 15129.751} C_VEL
LIN {X 0,Y 401.459,Z 152.041,A -85,B 0,C 180,E1 15125.718,E2 15125.718} C_VEL
LIN {X 0,Y 401.462,Z 152.04,A -85,B 0,C 180,E1 15121.713,E2 15121.713} C_VEL
LIN {X 0,Y 401.465,Z 152.033,A -85,B 0,C 180,E1 15117.716,E2 15117.716} C_VEL
LIN {X 0,Y 401.468,Z 152.025,A -85,B 0,C 180,E1 15113.709,E2 15113.709} C_VEL
LIN {X 0,Y 401.47,Z 152.021,A -85,B 0,C 180,E1 15109.815,E2 15109.815} C_VEL
LIN {X 0,Y 401.471,Z 151.982,A -85,B 0,C 180,E1 15105.873,E2 15105.873} C_VEL
LIN {X 0,Y 401.479,Z 152.029,A -85,B 0,C 180,E1 15101.862,E2 15101.862} C_VEL
LIN {X 0,Y 401.478,Z 151.978,A -85,B 0,C 180,E1 15097.883,E2 15097.883} C_VEL
LIN {X 0,Y 401.562,Z 152.403,A -85,B 0,C 180,E1 15096.601,E2 15096.601} C_VEL
LIN {X 0,Y 402.957,Z 155.756,A -85,B 0,C 180,E1 15095.52,E2 15095.52} C_VEL
LIN {X 0,Y 404.932,Z 158.122,A -85,B 0,C 180,E1 15094.555,E2 15094.555} C_VEL
LIN {X 0,Y 406.874,Z 161.804,A -85,B 0,C 180,E1 15093.433,E2 15093.433} C_VEL
LIN {X 0,Y 408.063,Z 163.301,A -85,B 0,C 180,E1 15092.887,E2 15092.887} C_VEL
LIN {X 0,Y 410.142,Z 167.188,A -85,B 0,C 180,E1 15091.775,E2 15091.775} C_VEL
LIN {X 0,Y 411.276,Z 169.048,A -85,B 0,C 180,E1 15091.226,E2 15091.226} C_VEL
LIN {X 0,Y 413.852,Z 173.083,A -85,B 0,C 180,E1 15090.113,E2 15090.113} C_VEL
LIN {X 0,Y 417.898,Z 178.19,A -85,B 0,C 180,E1 15089.082,E2 15089.082} C_VEL
LIN {X 0,Y 427.886,Z 191.3,A -85,B 0,C 180,E1 15086.733,E2 15086.733} C_VEL
LIN {X 0,Y 438.279,Z 205.579,A -85,B 0,C 180,E1 15084.508,E2 15084.508} C_VEL
LIN {X 0,Y 449.317,Z 222.087,A -85,B 0,C 180,E1 15082.33,E2 15082.33} C_VEL
LIN {X 0,Y 452.651,Z 227.609,A -85,B 0,C 180,E1 15081.698,E2 15081.698} C_VEL
LIN {X 0,Y 444.168,Z 443.108,A -85,B 0,C 180,E1 15077.646,E2 15077.646} C_VEL
LIN {X 0,Y 441.36,Z 512.51,A -85,B 0,C 180,E1 15076.314,E2 15076.314} C_VEL
LIN {X 0,Y 439.415,Z 535.697,A -85,B 0,C 180,E1 15075.666,E2 15075.666} C_VEL
LIN {X 0,Y 436.927,Z 559.227,A -85,B 0,C 180,E1 15074.768,E2 15074.768} C_VEL
LIN {X 0,Y 434.297,Z 579.521,A -85,B 0,C 180,E1 15073.773,E2 15073.773} C_VEL
LIN {X 0,Y 431.022,Z 601.409,A -85,B 0,C 180,E1 15072.456,E2 15072.456} C_VEL
LIN {X 0,Y 427.793,Z 620.8,A -85,B 0,C 180,E1 15071.052,E2 15071.052} C_VEL
LIN {X 0,Y 424.05,Z 641.406,A -85,B 0,C 180,E1 15069.277,E2 15069.277} C_VEL
LIN {X 0,Y 420.424,Z 660.671,A -85,B 0,C 180,E1 15067.332,E2 15067.332} C_VEL
LIN {X 0,Y 416.767,Z 678.969,A -85,B 0,C 180,E1 15065.153,E2 15065.153} C_VEL
LIN {X 0,Y 413.01,Z 698.095,A -85,B 0,C 180,E1 15062.509,E2 15062.509} C_VEL
LIN {X 0,Y 409.999,Z 713.806,A -85,B 0,C 180,E1 15059.994,E2 15059.994} C_VEL
LIN {X 0,Y 407.304,Z 728.114,A -85,B 0,C 180,E1 15057.297,E2 15057.297} C_VEL
LIN {X 0,Y 405.071,Z 740.993,A -85,B 0,C 180,E1 15054.499,E2 15054.499} C_VEL
LIN {X 0,Y 403.261,Z 752.219,A -85,B 0,C 180,E1 15051.599,E2 15051.599} C_VEL
LIN {X 0,Y 401.83,Z 762.581,A -85,B 0,C 180,E1 15048.421,E2 15048.421} C_VEL
LIN {X 0,Y 400.969,Z 770.113,A -85,B 0,C 180,E1 15045.623,E2 15045.623} C_VEL
LIN {X 0,Y 400.368,Z 777.189,A -85,B 0,C 180,E1 15042.402,E2 15042.402} C_VEL
LIN {X 0,Y 400.074,Z 782.054,A -85,B 0,C 180,E1 15039.494,E2 15039.494} C_VEL
LIN {X 0,Y 399.944,Z 785.969,A -85,B 0,C 180,E1 15036.315,E2 15036.315} C_VEL
LIN {X 0,Y 399.91,Z 788.108,A -85,B 0,C 180,E1 15033.297,E2 15033.297} C_VEL
LIN {X 0,Y 399.9,Z 788.938,A -85,B 0,C 180,E1 15030.43,E2 15030.43} C_VEL
LIN {X 0,Y 399.911,Z 788.385,A -85,B 0,C 180,E1 15027.277,E2 15027.277} C_VEL
LIN {X 0,Y 399.922,Z 786.673,A -85,B 0,C 180,E1 15024.549,E2 15024.549} C_VEL
LIN {X 0,Y 400.013,Z 783.527,A -85,B 0,C 180,E1 15021.52,E2 15021.52} C_VEL
LIN {X 0,Y 400.259,Z 778.772,A -85,B 0,C 180,E1 15018.473,E2 15018.473} C_VEL
LIN {X 0,Y 400.739,Z 772.602,A -85,B 0,C 180,E1 15015.405,E2 15015.405} C_VEL
LIN {X 0,Y 401.571,Z 764.695,A -85,B 0,C 180,E1 15012.317,E2 15012.317} C_VEL
LIN {X 0,Y 402.858,Z 755.13,A -85,B 0,C 180,E1 15009.212,E2 15009.212} C_VEL
LIN {X 0,Y 404.556,Z 744.008,A -85,B 0,C 180,E1 15006.244,E2 15006.244} C_VEL
LIN {X 0,Y 406.686,Z 731.682,A -85,B 0,C 180,E1 15003.42,E2 15003.42} C_VEL
LIN {X 0,Y 409.234,Z 717.763,A -85,B 0,C 180,E1 15000.719,E2 15000.719} C_VEL
LIN {X 0,Y 412.441,Z 701.034,A -85,B 0,C 180,E1 14997.934,E2 14997.934} C_VEL
LIN {X 0,Y 415.893,Z 683.577,A -85,B 0,C 180,E1 14995.434,E2 14995.434} C_VEL
LIN {X 0,Y 419.51,Z 665.084,A -85,B 0,C 180,E1 14993.173,E2 14993.173} C_VEL
LIN {X 0,Y 423.509,Z 644.344,A -85,B 0,C 180,E1 14991.003,E2 14991.003} C_VEL
LIN {X 0,Y 427.172,Z 624.397,A -85,B 0,C 180,E1 14989.23,E2 14989.23} C_VEL
LIN {X 0,Y 430.674,Z 603.442,A -85,B 0,C 180,E1 14987.682,E2 14987.682} C_VEL
LIN {X 0,Y 434.043,Z 581.415,A -85,B 0,C 180,E1 14986.33,E2 14986.33} C_VEL
LIN {X 0,Y 436.644,Z 561.424,A -85,B 0,C 180,E1 14985.334,E2 14985.334} C_VEL
LIN {X 0,Y 439.194,Z 538.162,A -85,B 0,C 180,E1 14984.418,E2 14984.418} C_VEL
LIN {X 0,Y 441.056,Z 516.214,A -85,B 0,C 180,E1 14983.779,E2 14983.779} C_VEL
LIN {X 0,Y 442.637,Z 483.398,A -85,B 0,C 180,E1 14983.112,E2 14983.112} C_VEL
LIN {X 0,Y 450.776,Z 274.163,A -85,B 0,C 180,E1 14979.177,E2 14979.177} C_VEL
LIN {X 0,Y 452.537,Z 227.132,A -85,B 0,C 180,E1 14978.278,E2 14978.278} C_VEL
LIN {X 0,Y 441.224,Z 209.892,A -85,B 0,C 180,E1 14976.099,E2 14976.099} C_VEL
LIN {X 0,Y 429.791,Z 193.724,A -85,B 0,C 180,E1 14973.7,E2 14973.7} C_VEL
LIN {X 0,Y 421.011,Z 182.378,A -85,B 0,C 180,E1 14971.698,E2 14971.698} C_VEL
LIN {X 0,Y 417.089,Z 177.383,A -85,B 0,C 180,E1 14970.744,E2 14970.744} C_VEL
LIN {X 0,Y 413.256,Z 172.452,A -85,B 0,C 180,E1 14969.735,E2 14969.735} C_VEL
LIN {X 0,Y 410.405,Z 167.499,A -85,B 0,C 180,E1 14968.364,E2 14968.364} C_VEL
LIN {X 0,Y 408.177,Z 163.674,A -85,B 0,C 180,E1 14967.231,E2 14967.231} C_VEL
LIN {X 0,Y 407.437,Z 162.4,A -85,B 0,C 180,E1 14966.842,E2 14966.842} C_VEL
LIN {X 0,Y 405.26,Z 159.129,A -85,B 0,C 180,E1 14965.736,E2 14965.736} C_VEL
LIN {X 0,Y 404.36,Z 157.214,A -85,B 0,C 180,E1 14965.17,E2 14965.17} C_VEL
LIN {X 0,Y 402.181,Z 154.432,A -85,B 0,C 180,E1 14964.061,E2 14964.061} C_VEL
LIN {X 0,Y 401.529,Z 152.195,A -85,B 0,C 180,E1 14963.324,E2 14963.324} C_VEL
LIN {X 0,Y 401.5,Z 152.006,A -85,B 0,C 180,E1 14959.493,E2 14959.493} C_VEL
LIN {X 0,Y 401.497,Z 151.968,A -85,B 0,C 180,E1 14955.454,E2 14955.454} C_VEL
LIN {X 0,Y 401.499,Z 152.028,A -85,B 0,C 180,E1 14951.491,E2 14951.491} C_VEL
LIN {X 0,Y 401.507,Z 152.02,A -85,B 0,C 180,E1 14947.44,E2 14947.44} C_VEL
LIN {X 0,Y 401.496,Z 152.02,A -85,B 0,C 180,E1 14943.426,E2 14943.426} C_VEL
LIN {X 0,Y 401.505,Z 152.019,A -85,B 0,C 180,E1 14939.429,E2 14939.429} C_VEL
LIN {X 0,Y 401.493,Z 152.023,A -85,B 0,C 180,E1 14935.429,E2 14935.429} C_VEL
LIN {X 0,Y 401.487,Z 152.03,A -85,B 0,C 180,E1 14931.551,E2 14931.551} C_VEL
LIN {X 0,Y 401.481,Z 152.038,A -85,B 0,C 180,E1 14927.633,E2 14927.633} C_VEL
LIN {X 0,Y 401.467,Z 152.04,A -85,B 0,C 180,E1 14923.803,E2 14923.803} C_VEL
LIN {X 0,Y 401.453,Z 151.981,A -85,B 0,C 180,E1 14919.897,E2 14919.897} C_VEL
LIN {X 0,Y 401.443,Z 152.001,A -85,B 0,C 180,E1 14916.203,E2 14916.203} C_VEL
LIN {X 0,Y 401.459,Z 152.12,A -85,B 0,C 180,E1 14914.319,E2 14914.319} C_VEL
LIN {X 0,Y 401.866,Z 153.701,A -85,B 0,C 180,E1 14913.713,E2 14913.713} C_VEL
LIN {X 0,Y 404.145,Z 157.088,A -85,B 0,C 180,E1 14912.442,E2 14912.442} C_VEL
LIN {X 0,Y 405.3,Z 159.406,A -85,B 0,C 180,E1 14911.724,E2 14911.724} C_VEL
LIN {X 0,Y 407.982,Z 163.572,A -85,B 0,C 180,E1 14910.327,E2 14910.327} C_VEL
LIN {X 0,Y 410.932,Z 168.781,A -85,B 0,C 180,E1 14908.784,E2 14908.784} C_VEL
LIN {X 0,Y 413.724,Z 173.825,A -85,B 0,C 180,E1 14907.389,E2 14907.389} C_VEL
LIN {X 0,Y 418.759,Z 182.99,A -85,B 0,C 180,E1 14905.037,E2 14905.037} C_VEL
LIN {X 0,Y 425.271,Z 195.843,A -85,B 0,C 180,E1 14902.147,E2 14902.147} C_VEL
LIN {X 0,Y 427.774,Z 200.667,A -85,B 0,C 180,E1 14901.214,E2 14901.214} C_VEL
LIN {X 0,Y 437.832,Z 215.621,A -85,B 0,C 180,E1 14899.071,E2 14899.071} C_VEL
LIN {X 0,Y 445.872,Z 228.578,A -85,B 0,C 180,E1 14897.47,E2 14897.47} C_VEL
LIN {X 0,Y 448.529,Z 249.473,A -85,B 0,C 180,E1 14896.578,E2 14896.578} C_VEL
LIN {X 0,Y 441.252,Z 477.311,A -85,B 0,C 180,E1 14892.592,E2 14892.592} C_VEL
LIN {X 0,Y 439.789,Z 518.208,A -85,B 0,C 180,E1 14891.85,E2 14891.85} C_VEL
LIN {X 0,Y 438.1,Z 539.57,A -85,B 0,C 180,E1 14891.26,E2 14891.26} C_VEL
LIN {X 0,Y 435.831,Z 560.982,A -85,B 0,C 180,E1 14890.436,E2 14890.436} C_VEL
LIN {X 0,Y 433.277,Z 580.408,A -85,B 0,C 180,E1 14889.475,E2 14889.475} C_VEL
LIN {X 0,Y 430.419,Z 598.365,A -85,B 0,C 180,E1 14888.367,E2 14888.367} C_VEL
LIN {X 0,Y 428.488,Z 605.357,A -85,B 0,C 180,E1 14887.977,E2 14887.977} C_VEL
LIN {X 0,Y 420.589,Z 622.727,A -85,B 0,C 180,E1 14887.139,E2 14887.139} C_VEL
LIN {X 0,Y 418.426,Z 629.194,A -85,B 0,C 180,E1 14886.639,E2 14886.639} C_VEL
LIN {X 0,Y 414.586,Z 646.737,A -85,B 0,C 180,E1 14884.859,E2 14884.859} C_VEL
LIN {X 0,Y 410.518,Z 664.375,A -85,B 0,C 180,E1 14882.731,E2 14882.731} C_VEL
LIN {X 0,Y 406.913,Z 679.583,A -85,B 0,C 180,E1 14880.572,E2 14880.572} C_VEL
LIN {X 0,Y 403.301,Z 694.519,A -85,B 0,C 180,E1 14878.043,E2 14878.043} C_VEL
LIN {X 0,Y 400.074,Z 708.2,A -85,B 0,C 180,E1 14875.299,E2 14875.299} C_VEL
LIN {X 0,Y 397.464,Z 720.064,A -85,B 0,C 180,E1 14872.48,E2 14872.48} C_VEL
LIN {X 0,Y 395.37,Z 730.475,A -85,B 0,C 180,E1 14869.5,E2 14869.5} C_VEL
LIN {X 0,Y 393.818,Z 739.434,A -85,B 0,C 180,E1 14866.368,E2 14866.368} C_VEL
LIN {X 0,Y 392.803,Z 746.989,A -85,B 0,C 180,E1 14863.093,E2 14863.093} C_VEL
LIN {X 0,Y 392.269,Z 752.539,A -85,B 0,C 180,E1 14859.981,E2 14859.981} C_VEL
LIN {X 0,Y 392.032,Z 756.503,A -85,B 0,C 180,E1 14856.884,E2 14856.884} C_VEL
LIN {X 0,Y 391.948,Z 759.091,A -85,B 0,C 180,E1 14853.803,E2 14853.803} C_VEL
LIN {X 0,Y 391.925,Z 760.108,A -85,B 0,C 180,E1 14850.731,E2 14850.731} C_VEL
LIN {X 0,Y 391.931,Z 759.717,A -85,B 0,C 180,E1 14847.514,E2 14847.514} C_VEL
LIN {X 0,Y 391.97,Z 757.977,A -85,B 0,C 180,E1 14844.584,E2 14844.584} C_VEL
LIN {X 0,Y 392.129,Z 754.517,A -85,B 0,C 180,E1 14841.348,E2 14841.348} C_VEL
LIN {X 0,Y 392.52,Z 749.76,A -85,B 0,C 180,E1 14838.242,E2 14838.242} C_VEL
LIN {X 0,Y 393.292,Z 743.096,A -85,B 0,C 180,E1 14835.032,E2 14835.032} C_VEL
LIN {X 0,Y 394.579,Z 734.785,A -85,B 0,C 180,E1 14831.84,E2 14831.84} C_VEL
LIN {X 0,Y 396.384,Z 725.318,A -85,B 0,C 180,E1 14828.857,E2 14828.857} C_VEL
LIN {X 0,Y 398.677,Z 714.418,A -85,B 0,C 180,E1 14826.029,E2 14826.029} C_VEL
LIN {X 0,Y 401.625,Z 701.558,A -85,B 0,C 180,E1 14823.218,E2 14823.218} C_VEL
LIN {X 0,Y 404.981,Z 687.599,A -85,B 0,C 180,E1 14820.636,E2 14820.636} C_VEL
LIN {X 0,Y 408.526,Z 672.792,A -85,B 0,C 180,E1 14818.334,E2 14818.334} C_VEL
LIN {X 0,Y 412.485,Z 655.979,A -85,B 0,C 180,E1 14816.117,E2 14816.117} C_VEL
LIN {X 0,Y 416.367,Z 638.961,A -85,B 0,C 180,E1 14814.217,E2 14814.217} C_VEL
LIN {X 0,Y 420.078,Z 621.016,A -85,B 0,C 180,E1 14812.547,E2 14812.547} C_VEL
LIN {X 0,Y 423.945,Z 600.61,A -85,B 0,C 180,E1 14810.973,E2 14810.973} C_VEL
LIN {X 0,Y 427.288,Z 580.635,A -85,B 0,C 180,E1 14809.716,E2 14809.716} C_VEL
LIN {X 0,Y 430.028,Z 560.617,A -85,B 0,C 180,E1 14808.721,E2 14808.721} C_VEL
LIN {X 0,Y 432.469,Z 538.201,A -85,B 0,C 180,E1 14807.864,E2 14807.864} C_VEL
LIN {X 0,Y 434.24,Z 516.36,A -85,B 0,C 180,E1 14807.275,E2 14807.275} C_VEL
LIN {X 0,Y 437.373,Z 423.466,A -85,B 0,C 180,E1 14805.626,E2 14805.626} C_VEL
LIN {X 0,Y 443.307,Z 249.784,A -85,B 0,C 180,E1 14802.538,E2 14802.538} C_VEL
LIN {X 0,Y 440.957,Z 232.657,A -85,B 0,C 180,E1 14801.757,E2 14801.757} C_VEL
LIN {X 0,Y 428.87,Z 213.585,A -85,B 0,C 180,E1 14799.227,E2 14799.227} C_VEL
LIN {X 0,Y 418.595,Z 198.624,A -85,B 0,C 180,E1 14796.837,E2 14796.837} C_VEL
LIN {X 0,Y 412.812,Z 187.305,A -85,B 0,C 180,E1 14794.189,E2 14794.189} C_VEL
LIN {X 0,Y 409.575,Z 181.47,A -85,B 0,C 180,E1 14792.65,E2 14792.65} C_VEL
LIN {X 0,Y 407.645,Z 177.806,A -85,B 0,C 180,E1 14791.661,E2 14791.661} C_VEL
LIN {X 0,Y 405.222,Z 173.361,A -85,B 0,C 180,E1 14790.386,E2 14790.386} C_VEL
LIN {X 0,Y 402.619,Z 168.732,A -85,B 0,C 180,E1 14788.964,E2 14788.964} C_VEL
LIN {X 0,Y 400.32,Z 164.926,A -85,B 0,C 180,E1 14787.682,E2 14787.682} C_VEL
LIN {X 0,Y 399.625,Z 163.6,A -85,B 0,C 180,E1 14787.25,E2 14787.25} C_VEL
LIN {X 0,Y 397.183,Z 159.768,A -85,B 0,C 180,E1 14785.818,E2 14785.818} C_VEL
LIN {X 0,Y 396.326,Z 158.133,A -85,B 0,C 180,E1 14785.237,E2 14785.237} C_VEL
LIN {X 0,Y 393.965,Z 154.853,A -85,B 0,C 180,E1 14783.799,E2 14783.799} C_VEL
LIN {X 0,Y 393.542,Z 153.143,A -85,B 0,C 180,E1 14783.119,E2 14783.119} C_VEL
LIN {X 0,Y 393.512,Z 152.962,A -85,B 0,C 180,E1 14779.288,E2 14779.288} C_VEL
LIN {X 0,Y 393.513,Z 153.025,A -85,B 0,C 180,E1 14775.474,E2 14775.474} C_VEL
LIN {X 0,Y 393.515,Z 153.018,A -85,B 0,C 180,E1 14771.58,E2 14771.58} C_VEL
LIN {X 0,Y 393.516,Z 153.014,A -85,B 0,C 180,E1 14767.593,E2 14767.593} C_VEL
LIN {X 0,Y 393.52,Z 153.012,A -85,B 0,C 180,E1 14763.642,E2 14763.642} C_VEL
LIN {X 0,Y 393.522,Z 153.014,A -85,B 0,C 180,E1 14759.709,E2 14759.709} C_VEL
LIN {X 0,Y 393.528,Z 153.017,A -85,B 0,C 180,E1 14755.775,E2 14755.775} C_VEL
LIN {X 0,Y 393.531,Z 153.022,A -85,B 0,C 180,E1 14751.82,E2 14751.82} C_VEL
LIN {X 0,Y 393.536,Z 153.026,A -85,B 0,C 180,E1 14747.826,E2 14747.826} C_VEL
LIN {X 0,Y 393.532,Z 152.963,A -85,B 0,C 180,E1 14743.771,E2 14743.771} C_VEL
LIN {X 0,Y 393.536,Z 152.977,A -85,B 0,C 180,E1 14739.786,E2 14739.786} C_VEL
LIN {X 0,Y 393.637,Z 153.47,A -85,B 0,C 180,E1 14739.014,E2 14739.014} C_VEL
LIN {X 0,Y 395.267,Z 157.026,A -85,B 0,C 180,E1 14737.701,E2 14737.701} C_VEL
LIN {X 0,Y 397.097,Z 159.148,A -85,B 0,C 180,E1 14736.715,E2 14736.715} C_VEL
LIN {X 0,Y 398.819,Z 162.655,A -85,B 0,C 180,E1 14735.565,E2 14735.565} C_VEL
LIN {X 0,Y 400.263,Z 164.24,A -85,B 0,C 180,E1 14734.871,E2 14734.871} C_VEL
LIN {X 0,Y 402.127,Z 167.992,A -85,B 0,C 180,E1 14733.731,E2 14733.731} C_VEL
LIN {X 0,Y 403.526,Z 170.005,A -85,B 0,C 180,E1 14733.036,E2 14733.036} C_VEL
LIN {X 0,Y 406.006,Z 174.033,A -85,B 0,C 180,E1 14731.862,E2 14731.862} C_VEL
LIN {X 0,Y 410.811,Z 179.844,A -85,B 0,C 180,E1 14730.552,E2 14730.552} C_VEL
LIN {X 0,Y 420.183,Z 191.999,A -85,B 0,C 180,E1 14728.192,E2 14728.192} C_VEL
LIN {X 0,Y 430.758,Z 206.278,A -85,B 0,C 180,E1 14725.785,E2 14725.785} C_VEL
LIN {X 0,Y 442.048,Z 222.892,A -85,B 0,C 180,E1 14723.436,E2 14723.436} C_VEL
LIN {X 0,Y 447.281,Z 231.405,A -85,B 0,C 180,E1 14722.404,E2 14722.404} C_VEL
LIN {X 0,Y 438.444,Z 445.652,A -85,B 0,C 180,E1 14718.341,E2 14718.341} C_VEL
LIN {X 0,Y 435.591,Z 512.743,A -85,B 0,C 180,E1 14717.039,E2 14717.039} C_VEL
LIN {X 0,Y 433.556,Z 535.958,A -85,B 0,C 180,E1 14716.384,E2 14716.384} C_VEL
LIN {X 0,Y 430.927,Z 559.628,A -85,B 0,C 180,E1 14715.469,E2 14715.469} C_VEL
LIN {X 0,Y 428.184,Z 579.843,A -85,B 0,C 180,E1 14714.468,E2 14714.468} C_VEL
LIN {X 0,Y 424.757,Z 601.676,A -85,B 0,C 180,E1 14713.137,E2 14713.137} C_VEL
LIN {X 0,Y 421.388,Z 620.956,A -85,B 0,C 180,E1 14711.724,E2 14711.724} C_VEL
LIN {X 0,Y 417.454,Z 641.476,A -85,B 0,C 180,E1 14709.932,E2 14709.932} C_VEL
LIN {X 0,Y 413.645,Z 660.601,A -85,B 0,C 180,E1 14707.972,E2 14707.972} C_VEL
LIN {X 0,Y 409.822,Z 678.71,A -85,B 0,C 180,E1 14705.779,E2 14705.779} C_VEL
LIN {X 0,Y 405.993,Z 696.871,A -85,B 0,C 180,E1 14703.226,E2 14703.226} C_VEL
LIN {X 0,Y 402.682,Z 712.975,A -85,B 0,C 180,E1 14700.597,E2 14700.597} C_VEL
LIN {X 0,Y 399.845,Z 727.274,A -85,B 0,C 180,E1 14697.879,E2 14697.879} C_VEL
LIN {X 0,Y 397.439,Z 740.378,A -85,B 0,C 180,E1 14695.001,E2 14695.001} C_VEL
LIN {X 0,Y 395.554,Z 751.381,A -85,B 0,C 180,E1 14692.125,E2 14692.125} C_VEL
LIN {X 0,Y 394.1,Z 761.304,A -85,B 0,C 180,E1 14689.103,E2 14689.103} C_VEL
LIN {X 0,Y 393.089,Z 769.353,A -85,B 0,C 180,E1 14686.096,E2 14686.096} C_VEL
LIN {X 0,Y 392.442,Z 776.303,A -85,B 0,C 180,E1 14682.956,E2 14682.956} C_VEL
LIN {X 0,Y 392.091,Z 781.506,A -85,B 0,C 180,E1 14679.837,E2 14679.837} C_VEL
LIN {X 0,Y 391.965,Z 785.193,A -85,B 0,C 180,E1 14676.886,E2 14676.886} C_VEL
LIN {X 0,Y 391.915,Z 787.671,A -85,B 0,C 180,E1 14673.657,E2 14673.657} C_VEL
LIN {X 0,Y 391.911,Z 788.59,A -85,B 0,C 180,E1 14670.877,E2 14670.877} C_VEL
LIN {X 0,Y 391.911,Z 788.303,A -85,B 0,C 180,E1 14667.661,E2 14667.661} C_VEL
LIN {X 0,Y 391.924,Z 786.488,A -85,B 0,C 180,E1 14664.584,E2 14664.584} C_VEL
LIN {X 0,Y 392.013,Z 783.542,A -85,B 0,C 180,E1 14661.641,E2 14661.641} C_VEL
LIN {X 0,Y 392.268,Z 778.689,A -85,B 0,C 180,E1 14658.384,E2 14658.384} C_VEL
LIN {X 0,Y 392.738,Z 772.856,A -85,B 0,C 180,E1 14655.402,E2 14655.402} C_VEL
LIN {X 0,Y 393.647,Z 764.686,A -85,B 0,C 180,E1 14652.102,E2 14652.102} C_VEL
LIN {X 0,Y 394.908,Z 755.67,A -85,B 0,C 180,E1 14649.108,E2 14649.108} C_VEL
LIN {X 0,Y 396.683,Z 744.612,A -85,B 0,C 180,E1 14646.059,E2 14646.059} C_VEL
LIN {X 0,Y 398.911,Z 732.319,A -85,B 0,C 180,E1 14643.163,E2 14643.163} C_VEL
LIN {X 0,Y 401.512,Z 718.754,A -85,B 0,C 180,E1 14640.459,E2 14640.459} C_VEL
LIN {X 0,Y 404.701,Z 703.15,A -85,B 0,C 180,E1 14637.749,E2 14637.749} C_VEL
LIN {X 0,Y 408.184,Z 686.496,A -85,B 0,C 180,E1 14635.265,E2 14635.265} C_VEL
LIN {X 0,Y 412.146,Z 667.569,A -85,B 0,C 180,E1 14632.839,E2 14632.839} C_VEL
LIN {X 0,Y 416.017,Z 648.97,A -85,B 0,C 180,E1 14630.796,E2 14630.796} C_VEL
LIN {X 0,Y 419.745,Z 629.585,A -85,B 0,C 180,E1 14628.995,E2 14628.995} C_VEL
LIN {X 0,Y 423.543,Z 608.771,A -85,B 0,C 180,E1 14627.351,E2 14627.351} C_VEL
LIN {X 0,Y 426.884,Z 588.309,A -85,B 0,C 180,E1 14626.016,E2 14626.016} C_VEL
LIN {X 0,Y 430.186,Z 565.345,A -85,B 0,C 180,E1 14624.797,E2 14624.797} C_VEL
LIN {X 0,Y 432.619,Z 545.232,A -85,B 0,C 180,E1 14623.947,E2 14623.947} C_VEL
LIN {X 0,Y 434.861,Z 521.772,A -85,B 0,C 180,E1 14623.198,E2 14623.198} C_VEL
LIN {X 0,Y 436.355,Z 498.276,A -85,B 0,C 180,E1 14622.659,E2 14622.659} C_VEL
LIN {X 0,Y 444.899,Z 287.859,A -85,B 0,C 180,E1 14618.667,E2 14618.667} C_VEL
LIN {X 0,Y 447.125,Z 230.84,A -85,B 0,C 180,E1 14617.563,E2 14617.563} C_VEL
LIN {X 0,Y 435.477,Z 213.034,A -85,B 0,C 180,E1 14615.231,E2 14615.231} C_VEL
LIN {X 0,Y 424.777,Z 198.134,A -85,B 0,C 180,E1 14612.898,E2 14612.898} C_VEL
LIN {X 0,Y 417.537,Z 188.629,A -85,B 0,C 180,E1 14611.188,E2 14611.188} C_VEL
LIN {X 0,Y 413.792,Z 183.839,A -85,B 0,C 180,E1 14610.252,E2 14610.252} C_VEL
LIN {X 0,Y 409.785,Z 178.837,A -85,B 0,C 180,E1 14609.208,E2 14609.208} C_VEL
LIN {X 0,Y 405.493,Z 173.501,A -85,B 0,C 180,E1 14608.017,E2 14608.017} C_VEL
LIN {X 0,Y 402.977,Z 168.956,A -85,B 0,C 180,E1 14606.685,E2 14606.685} C_VEL
LIN {X 0,Y 400.581,Z 165.235,A -85,B 0,C 180,E1 14605.424,E2 14605.424} C_VEL
LIN {X 0,Y 399.922,Z 163.795,A -85,B 0,C 180,E1 14604.994,E2 14604.994} C_VEL
LIN {X 0,Y 397.569,Z 160.546,A -85,B 0,C 180,E1 14603.727,E2 14603.727} C_VEL
LIN {X 0,Y 396.557,Z 158.301,A -85,B 0,C 180,E1 14603.005,E2 14603.005} C_VEL
LIN {X 0,Y 394.305,Z 155.49,A -85,B 0,C 180,E1 14601.729,E2 14601.729} C_VEL
LIN {X 0,Y 393.595,Z 153.25,A -85,B 0,C 180,E1 14600.911,E2 14600.911} C_VEL
LIN {X 0,Y 393.558,Z 152.979,A -85,B 0,C 180,E1 14597.14,E2 14597.14} C_VEL
LIN {X 0,Y 393.563,Z 152.986,A -85,B 0,C 180,E1 14593.217,E2 14593.217} C_VEL
LIN {X 0,Y 393.565,Z 153.014,A -85,B 0,C 180,E1 14589.21,E2 14589.21} C_VEL
LIN {X 0,Y 393.564,Z 153.024,A -85,B 0,C 180,E1 14585.218,E2 14585.218} C_VEL
LIN {X 0,Y 393.567,Z 153.021,A -85,B 0,C 180,E1 14581.164,E2 14581.164} C_VEL
LIN {X 0,Y 393.56,Z 153.015,A -85,B 0,C 180,E1 14577.233,E2 14577.233} C_VEL
LIN {X 0,Y 393.567,Z 153.009,A -85,B 0,C 180,E1 14573.142,E2 14573.142} C_VEL
LIN {X 0,Y 393.554,Z 153.009,A -85,B 0,C 180,E1 14569.163,E2 14569.163} C_VEL
LIN {X 0,Y 393.559,Z 153.011,A -85,B 0,C 180,E1 14565.132,E2 14565.132} C_VEL
LIN {X 0,Y 393.546,Z 152.96,A -85,B 0,C 180,E1 14561.176,E2 14561.176} C_VEL
LIN {X 0,Y 393.554,Z 153.023,A -85,B 0,C 180,E1 14557.126,E2 14557.126} C_VEL
LIN {X 0,Y 393.6,Z 153.554,A -85,B 0,C 180,E1 14556.494,E2 14556.494} C_VEL
LIN {X 0,Y 395.291,Z 157.049,A -85,B 0,C 180,E1 14555.173,E2 14555.173} C_VEL
LIN {X 0,Y 397.047,Z 159.325,A -85,B 0,C 180,E1 14554.173,E2 14554.173} C_VEL
LIN {X 0,Y 399.093,Z 163.042,A -85,B 0,C 180,E1 14552.872,E2 14552.872} C_VEL
LIN {X 0,Y 400.171,Z 164.478,A -85,B 0,C 180,E1 14552.307,E2 14552.307} C_VEL
LIN {X 0,Y 402.458,Z 168.554,A -85,B 0,C 180,E1 14550.983,E2 14550.983} C_VEL
LIN {X 0,Y 406.293,Z 175.388,A -85,B 0,C 180,E1 14548.912,E2 14548.912} C_VEL
LIN {X 0,Y 409.108,Z 180.546,A -85,B 0,C 180,E1 14547.474,E2 14547.474} C_VEL
LIN {X 0,Y 413.538,Z 188.54,A -85,B 0,C 180,E1 14545.376,E2 14545.376} C_VEL
LIN {X 0,Y 419.201,Z 199.569,A -85,B 0,C 180,E1 14542.883,E2 14542.883} C_VEL
LIN {X 0,Y 429.851,Z 215.242,A -85,B 0,C 180,E1 14540.449,E2 14540.449} C_VEL
LIN {X 0,Y 441.031,Z 232.857,A -85,B 0,C 180,E1 14538.124,E2 14538.124} C_VEL
LIN {X 0,Y 443.265,Z 251.075,A -85,B 0,C 180,E1 14537.335,E2 14537.335} C_VEL
LIN {X 0,Y 435.558,Z 479.649,A -85,B 0,C 180,E1 14533.299,E2 14533.299} C_VEL
LIN {X 0,Y 434.086,Z 518.266,A -85,B 0,C 180,E1 14532.589,E2 14532.589} C_VEL
LIN {X 0,Y 432.324,Z 539.629,A -85,B 0,C 180,E1 14531.997,E2 14531.997} C_VEL
LIN {X 0,Y 429.93,Z 561.242,A -85,B 0,C 180,E1 14531.158,E2 14531.158} C_VEL
LIN {X 0,Y 427.17,Z 581.327,A -85,B 0,C 180,E1 14530.153,E2 14530.153} C_VEL
LIN {X 0,Y 423.947,Z 600.48,A -85,B 0,C 180,E1 14528.944,E2 14528.944} C_VEL
LIN {X 0,Y 420.245,Z 620.139,A -85,B 0,C 180,E1 14527.436,E2 14527.436} C_VEL
LIN {X 0,Y 418.426,Z 629.194,A -85,B 0,C 180,E1 14526.639,E2 14526.639} C_VEL
LIN {X 0,Y 416.213,Z 635.678,A -85,B 0,C 180,E1 14526.104,E2 14526.104} C_VEL
LIN {X 0,Y 407.732,Z 651.8,A -85,B 0,C 180,E1 14524.91,E2 14524.91} C_VEL
LIN {X 0,Y 405.508,Z 657.612,A -85,B 0,C 180,E1 14524.292,E2 14524.292} C_VEL
LIN {X 0,Y 401.378,Z 674.199,A -85,B 0,C 180,E1 14522.045,E2 14522.045} C_VEL
LIN {X 0,Y 397.658,Z 688.968,A -85,B 0,C 180,E1 14519.691,E2 14519.691} C_VEL
LIN {X 0,Y 394.167,Z 702.711,A -85,B 0,C 180,E1 14517.081,E2 14517.081} C_VEL
LIN {X 0,Y 391.001,Z 715.715,A -85,B 0,C 180,E1 14514.151,E2 14514.151} C_VEL
LIN {X 0,Y 388.495,Z 726.962,A -85,B 0,C 180,E1 14511.119,E2 14511.119} C_VEL
LIN {X 0,Y 386.647,Z 736.266,A -85,B 0,C 180,E1 14508.078,E2 14508.078} C_VEL
LIN {X 0,Y 385.338,Z 744.186,A -85,B 0,C 180,E1 14504.885,E2 14504.885} C_VEL
LIN {X 0,Y 384.55,Z 750.486,A -85,B 0,C 180,E1 14501.701,E2 14501.701} C_VEL
LIN {X 0,Y 384.15,Z 755.199,A -85,B 0,C 180,E1 14498.483,E2 14498.483} C_VEL
LIN {X 0,Y 383.978,Z 758.44,A -85,B 0,C 180,E1 14495.229,E2 14495.229} C_VEL
LIN {X 0,Y 383.937,Z 760.168,A -85,B 0,C 180,E1 14492.089,E2 14492.089} C_VEL
LIN {X 0,Y 383.939,Z 760.368,A -85,B 0,C 180,E1 14488.955,E2 14488.955} C_VEL
LIN {X 0,Y 383.962,Z 759.262,A -85,B 0,C 180,E1 14485.819,E2 14485.819} C_VEL
LIN {X 0,Y 384.061,Z 756.612,A -85,B 0,C 180,E1 14482.671,E2 14482.671} C_VEL
LIN {X 0,Y 384.364,Z 752.317,A -85,B 0,C 180,E1 14479.357,E2 14479.357} C_VEL
LIN {X 0,Y 385.006,Z 746.693,A -85,B 0,C 180,E1 14476.177,E2 14476.177} C_VEL
LIN {X 0,Y 386.108,Z 739.314,A -85,B 0,C 180,E1 14472.985,E2 14472.985} C_VEL
LIN {X 0,Y 387.919,Z 729.705,A -85,B 0,C 180,E1 14469.638,E2 14469.638} C_VEL
LIN {X 0,Y 390.244,Z 719.11,A -85,B 0,C 180,E1 14466.602,E2 14466.602} C_VEL
LIN {X 0,Y 393.106,Z 706.997,A -85,B 0,C 180,E1 14463.733,E2 14463.733} C_VEL
LIN {X 0,Y 396.477,Z 693.511,A -85,B 0,C 180,E1 14461.041,E2 14461.041} C_VEL
LIN {X 0,Y 400.212,Z 678.979,A -85,B 0,C 180,E1 14458.576,E2 14458.576} C_VEL
LIN {X 0,Y 404.116,Z 663.318,A -85,B 0,C 180,E1 14456.344,E2 14456.344} C_VEL
LIN {X 0,Y 408.285,Z 646.056,A -85,B 0,C 180,E1 14454.264,E2 14454.264} C_VEL
LIN {X 0,Y 412.371,Z 628.245,A -85,B 0,C 180,E1 14452.454,E2 14452.454} C_VEL
LIN {X 0,Y 416.162,Z 609.716,A -85,B 0,C 180,E1 14450.899,E2 14450.899} C_VEL
LIN {X 0,Y 419.966,Z 588.93,A -85,B 0,C 180,E1 14449.463,E2 14449.463} C_VEL
LIN {X 0,Y 423.143,Z 568.902,A -85,B 0,C 180,E1 14448.347,E2 14448.347} C_VEL
LIN {X 0,Y 425.7,Z 548.574,A -85,B 0,C 180,E1 14447.473,E2 14447.473} C_VEL
LIN {X 0,Y 427.857,Z 526.526,A -85,B 0,C 180,E1 14446.766,E2 14446.766} C_VEL
LIN {X 0,Y 429.215,Z 504.433,A -85,B 0,C 180,E1 14446.279,E2 14446.279} C_VEL
LIN {X 0,Y 437.051,Z 280.071,A -85,B 0,C 180,E1 14442.29,E2 14442.29} C_VEL
LIN {X 0,Y 438.059,Z 250.923,A -85,B 0,C 180,E1 14441.74,E2 14441.74} C_VEL
LIN {X 0,Y 436.194,Z 237.136,A -85,B 0,C 180,E1 14441.094,E2 14441.094} C_VEL
LIN {X 0,Y 424.805,Z 219.074,A -85,B 0,C 180,E1 14438.632,E2 14438.632} C_VEL
LIN {X 0,Y 414.516,Z 203.989,A -85,B 0,C 180,E1 14436.183,E2 14436.183} C_VEL
LIN {X 0,Y 409.984,Z 197.425,A -85,B 0,C 180,E1 14434.968,E2 14434.968} C_VEL
LIN {X 0,Y 404.993,Z 188.118,A -85,B 0,C 180,E1 14432.562,E2 14432.562} C_VEL
LIN {X 0,Y 402.51,Z 183.494,A -85,B 0,C 180,E1 14431.277,E2 14431.277} C_VEL
LIN {X 0,Y 400.12,Z 179.11,A -85,B 0,C 180,E1 14429.986,E2 14429.986} C_VEL
LIN {X 0,Y 397.83,Z 174.944,A -85,B 0,C 180,E1 14428.688,E2 14428.688} C_VEL
LIN {X 0,Y 394.875,Z 169.858,A -85,B 0,C 180,E1 14426.952,E2 14426.952} C_VEL
LIN {X 0,Y 392.547,Z 165.901,A -85,B 0,C 180,E1 14425.497,E2 14425.497} C_VEL
LIN {X 0,Y 391.623,Z 164.449,A -85,B 0,C 180,E1 14424.915,E2 14424.915} C_VEL
LIN {X 0,Y 389.409,Z 160.994,A -85,B 0,C 180,E1 14423.452,E2 14423.452} C_VEL
LIN {X 0,Y 388.707,Z 159.387,A -85,B 0,C 180,E1 14422.856,E2 14422.856} C_VEL
LIN {X 0,Y 386.275,Z 156.398,A -85,B 0,C 180,E1 14421.247,E2 14421.247} C_VEL
LIN {X 0,Y 385.627,Z 154.259,A -85,B 0,C 180,E1 14420.331,E2 14420.331} C_VEL
LIN {X 0,Y 385.594,Z 153.98,A -85,B 0,C 180,E1 14417.039,E2 14417.039} C_VEL
LIN {X 0,Y 385.59,Z 154.009,A -85,B 0,C 180,E1 14413.191,E2 14413.191} C_VEL
LIN {X 0,Y 385.592,Z 154.018,A -85,B 0,C 180,E1 14409.252,E2 14409.252} C_VEL
LIN {X 0,Y 385.593,Z 154.016,A -85,B 0,C 180,E1 14405.315,E2 14405.315} C_VEL
LIN {X 0,Y 385.592,Z 154.008,A -85,B 0,C 180,E1 14401.337,E2 14401.337} C_VEL
LIN {X 0,Y 385.591,Z 154.005,A -85,B 0,C 180,E1 14397.474,E2 14397.474} C_VEL
LIN {X 0,Y 385.594,Z 153.999,A -85,B 0,C 180,E1 14393.449,E2 14393.449} C_VEL
LIN {X 0,Y 385.594,Z 153.997,A -85,B 0,C 180,E1 14389.542,E2 14389.542} C_VEL
LIN {X 0,Y 385.592,Z 153.95,A -85,B 0,C 180,E1 14385.586,E2 14385.586} C_VEL
LIN {X 0,Y 385.64,Z 154.25,A -85,B 0,C 180,E1 14382.029,E2 14382.029} C_VEL
LIN {X 0,Y 387.269,Z 157.938,A -85,B 0,C 180,E1 14380.389,E2 14380.389} C_VEL
LIN {X 0,Y 389.198,Z 159.96,A -85,B 0,C 180,E1 14379.236,E2 14379.236} C_VEL
LIN {X 0,Y 390.905,Z 163.582,A -85,B 0,C 180,E1 14377.914,E2 14377.914} C_VEL
LIN {X 0,Y 392.669,Z 165.791,A -85,B 0,C 180,E1 14376.913,E2 14376.913} C_VEL
LIN {X 0,Y 394.682,Z 169.535,A -85,B 0,C 180,E1 14375.611,E2 14375.611} C_VEL
LIN {X 0,Y 395.775,Z 170.917,A -85,B 0,C 180,E1 14375.046,E2 14375.046} C_VEL
LIN {X 0,Y 398.084,Z 174.918,A -85,B 0,C 180,E1 14373.805,E2 14373.805} C_VEL
LIN {X 0,Y 400.195,Z 177.548,A -85,B 0,C 180,E1 14373.154,E2 14373.154} C_VEL
LIN {X 0,Y 404.619,Z 182.846,A -85,B 0,C 180,E1 14371.877,E2 14371.877} C_VEL
LIN {X 0,Y 409.31,Z 188.696,A -85,B 0,C 180,E1 14370.594,E2 14370.594} C_VEL
LIN {X 0,Y 414.16,Z 194.929,A -85,B 0,C 180,E1 14369.337,E2 14369.337} C_VEL
LIN {X 0,Y 423.809,Z 207.758,A -85,B 0,C 180,E1 14367.017,E2 14367.017} C_VEL
LIN {X 0,Y 435.326,Z 224.515,A -85,B 0,C 180,E1 14364.493,E2 14364.493} C_VEL
LIN {X 0,Y 441.984,Z 235.164,A -85,B 0,C 180,E1 14363.128,E2 14363.128} C_VEL
LIN {X 0,Y 432.792,Z 448.139,A -85,B 0,C 180,E1 14359.056,E2 14359.056} C_VEL
LIN {X 0,Y 429.911,Z 512.786,A -85,B 0,C 180,E1 14357.788,E2 14357.788} C_VEL
LIN {X 0,Y 427.782,Z 536.124,A -85,B 0,C 180,E1 14357.125,E2 14357.125} C_VEL
LIN {X 0,Y 424.998,Z 560.063,A -85,B 0,C 180,E1 14356.191,E2 14356.191} C_VEL
LIN {X 0,Y 422.049,Z 580.854,A -85,B 0,C 180,E1 14355.147,E2 14355.147} C_VEL
LIN {X 0,Y 418.52,Z 602.19,A -85,B 0,C 180,E1 14353.823,E2 14353.823} C_VEL
LIN {X 0,Y 414.835,Z 622.313,A -85,B 0,C 180,E1 14352.325,E2 14352.325} C_VEL
LIN {X 0,Y 410.765,Z 642.343,A -85,B 0,C 180,E1 14350.534,E2 14350.534} C_VEL
LIN {X 0,Y 406.614,Z 661.964,A -85,B 0,C 180,E1 14348.47,E2 14348.47} C_VEL
LIN {X 0,Y 402.771,Z 679.284,A -85,B 0,C 180,E1 14346.327,E2 14346.327} C_VEL
LIN {X 0,Y 398.739,Z 697.262,A -85,B 0,C 180,E1 14343.739,E2 14343.739} C_VEL
LIN {X 0,Y 395.255,Z 713.226,A -85,B 0,C 180,E1 14341.067,E2 14341.067} C_VEL
LIN {X 0,Y 392.1,Z 728.055,A -85,B 0,C 180,E1 14338.147,E2 14338.147} C_VEL
LIN {X 0,Y 389.429,Z 741.812,A -85,B 0,C 180,E1 14334.998,E2 14334.998} C_VEL
LIN {X 0,Y 387.554,Z 752.45,A -85,B 0,C 180,E1 14332.127,E2 14332.127} C_VEL
LIN {X 0,Y 386.005,Z 762.519,A -85,B 0,C 180,E1 14328.891,E2 14328.891} C_VEL
LIN {X 0,Y 385.056,Z 770.041,A -85,B 0,C 180,E1 14325.976,E2 14325.976} C_VEL
LIN {X 0,Y 384.396,Z 777.012,A -85,B 0,C 180,E1 14322.62,E2 14322.62} C_VEL
LIN {X 0,Y 384.085,Z 781.607,A -85,B 0,C 180,E1 14319.742,E2 14319.742} C_VEL
LIN {X 0,Y 383.952,Z 785.474,A -85,B 0,C 180,E1 14316.429,E2 14316.429} C_VEL
LIN {X 0,Y 383.918,Z 787.516,A -85,B 0,C 180,E1 14313.434,E2 14313.434} C_VEL
LIN {X 0,Y 383.911,Z 788.346,A -85,B 0,C 180,E1 14310.597,E2 14310.597} C_VEL
LIN {X 0,Y 383.919,Z 787.87,A -85,B 0,C 180,E1 14307.313,E2 14307.313} C_VEL
LIN {X 0,Y 383.929,Z 786.066,A -85,B 0,C 180,E1 14304.321,E2 14304.321} C_VEL
LIN {X 0,Y 384.027,Z 782.884,A -85,B 0,C 180,E1 14301.164,E2 14301.164} C_VEL
LIN {X 0,Y 384.315,Z 778.072,A -85,B 0,C 180,E1 14297.987,E2 14297.987} C_VEL
LIN {X 0,Y 384.871,Z 771.839,A -85,B 0,C 180,E1 14294.789,E2 14294.789} C_VEL
LIN {X 0,Y 385.853,Z 763.655,A -85,B 0,C 180,E1 14291.515,E2 14291.515} C_VEL
LIN {X 0,Y 387.304,Z 754.083,A -85,B 0,C 180,E1 14288.336,E2 14288.336} C_VEL
LIN {X 0,Y 389.25,Z 742.795,A -85,B 0,C 180,E1 14285.249,E2 14285.249} C_VEL
LIN {X 0,Y 391.809,Z 729.531,A -85,B 0,C 180,E1 14282.161,E2 14282.161} C_VEL
LIN {X 0,Y 394.7,Z 715.671,A -85,B 0,C 180,E1 14279.392,E2 14279.392} C_VEL
LIN {X 0,Y 398.209,Z 699.663,A -85,B 0,C 180,E1 14276.642,E2 14276.642} C_VEL
LIN {X 0,Y 401.903,Z 683.243,A -85,B 0,C 180,E1 14274.196,E2 14274.196} C_VEL
LIN {X 0,Y 405.908,Z 665.083,A -85,B 0,C 180,E1 14271.9,E2 14271.9} C_VEL
LIN {X 0,Y 410.149,Z 645.332,A -85,B 0,C 180,E1 14269.76,E2 14269.76} C_VEL
LIN {X 0,Y 414.008,Z 626.324,A -85,B 0,C 180,E1 14268.014,E2 14268.014} C_VEL
LIN {X 0,Y 418.017,Z 604.905,A -85,B 0,C 180,E1 14266.366,E2 14266.366} C_VEL
LIN {X 0,Y 421.584,Z 584.006,A -85,B 0,C 180,E1 14265.03,E2 14265.03} C_VEL
LIN {X 0,Y 424.692,Z 562.226,A -85,B 0,C 180,E1 14263.913,E2 14263.913} C_VEL
LIN {X 0,Y 427.414,Z 539.868,A -85,B 0,C 180,E1 14263.004,E2 14263.004} C_VEL
LIN {X 0,Y 429.481,Z 517.546,A -85,B 0,C 180,E1 14262.336,E2 14262.336} C_VEL
LIN {X 0,Y 431.196,Z 486.192,A -85,B 0,C 180,E1 14261.675,E2 14261.675} C_VEL
LIN {X 0,Y 440.093,Z 277.742,A -85,B 0,C 180,E1 14257.686,E2 14257.686} C_VEL
LIN {X 0,Y 441.844,Z 234.738,A -85,B 0,C 180,E1 14256.846,E2 14256.846} C_VEL
LIN {X 0,Y 430.994,Z 218.087,A -85,B 0,C 180,E1 14254.596,E2 14254.596} C_VEL
LIN {X 0,Y 419.746,Z 202.174,A -85,B 0,C 180,E1 14252.046,E2 14252.046} C_VEL
LIN {X 0,Y 410.766,Z 190.552,A -85,B 0,C 180,E1 14249.813,E2 14249.813} C_VEL
LIN {X 0,Y 406.699,Z 185.455,A -85,B 0,C 180,E1 14248.726,E2 14248.726} C_VEL
LIN {X 0,Y 402.535,Z 180.279,A -85,B 0,C 180,E1 14247.557,E2 14247.557} C_VEL
LIN {X 0,Y 397.975,Z 174.817,A -85,B 0,C 180,E1 14246.202,E2 14246.202} C_VEL
LIN {X 0,Y 395.726,Z 170.791,A -85,B 0,C 180,E1 14244.957,E2 14244.957} C_VEL
LIN {X 0,Y 392.964,Z 166.654,A -85,B 0,C 180,E1 14243.386,E2 14243.386} C_VEL
LIN {X 0,Y 392.157,Z 164.898,A -85,B 0,C 180,E1 14242.802,E2 14242.802} C_VEL
LIN {X 0,Y 389.774,Z 161.624,A -85,B 0,C 180,E1 14241.362,E2 14241.362} C_VEL
LIN {X 0,Y 388.898,Z 159.538,A -85,B 0,C 180,E1 14240.623,E2 14240.623} C_VEL
LIN {X 0,Y 386.226,Z 156.217,A -85,B 0,C 180,E1 14238.88,E2 14238.88} C_VEL
LIN {X 0,Y 385.627,Z 154.162,A -85,B 0,C 180,E1 14237.971,E2 14237.971} C_VEL
LIN {X 0,Y 385.594,Z 153.954,A -85,B 0,C 180,E1 14234.107,E2 14234.107} C_VEL
LIN {X 0,Y 385.597,Z 153.997,A -85,B 0,C 180,E1 14230.156,E2 14230.156} C_VEL
LIN {X 0,Y 385.594,Z 154.003,A -85,B 0,C 180,E1 14226.103,E2 14226.103} C_VEL
LIN {X 0,Y 385.592,Z 154.011,A -85,B 0,C 180,E1 14222.08,E2 14222.08} C_VEL
LIN {X 0,Y 385.591,Z 154.018,A -85,B 0,C 180,E1 14218.068,E2 14218.068} C_VEL
LIN {X 0,Y 385.587,Z 154.015,A -85,B 0,C 180,E1 14214.046,E2 14214.046} C_VEL
LIN {X 0,Y 385.582,Z 154.009,A -85,B 0,C 180,E1 14210.145,E2 14210.145} C_VEL
LIN {X 0,Y 385.576,Z 154.004,A -85,B 0,C 180,E1 14206.198,E2 14206.198} C_VEL
LIN {X 0,Y 385.57,Z 153.964,A -85,B 0,C 180,E1 14202.182,E2 14202.182} C_VEL
LIN {X 0,Y 385.64,Z 154.244,A -85,B 0,C 180,E1 14199.511,E2 14199.511} C_VEL
LIN {X 0,Y 387.245,Z 157.987,A -85,B 0,C 180,E1 14197.854,E2 14197.854} C_VEL
LIN {X 0,Y 389.132,Z 160.094,A -85,B 0,C 180,E1 14196.69,E2 14196.69} C_VEL
LIN {X 0,Y 390.89,Z 163.611,A -85,B 0,C 180,E1 14195.358,E2 14195.358} C_VEL
LIN {X 0,Y 392.415,Z 165.462,A -85,B 0,C 180,E1 14194.494,E2 14194.494} C_VEL
LIN {X 0,Y 394.642,Z 169.6,A -85,B 0,C 180,E1 14193.031,E2 14193.031} C_VEL
LIN {X 0,Y 395.653,Z 171.155,A -85,B 0,C 180,E1 14192.454,E2 14192.454} C_VEL
LIN {X 0,Y 398.647,Z 176.406,A -85,B 0,C 180,E1 14190.719,E2 14190.719} C_VEL
LIN {X 0,Y 401.517,Z 181.627,A -85,B 0,C 180,E1 14189.137,E2 14189.137} C_VEL
LIN {X 0,Y 406.27,Z 190.299,A -85,B 0,C 180,E1 14186.714,E2 14186.714} C_VEL
LIN {X 0,Y 410.71,Z 198.654,A -85,B 0,C 180,E1 14184.677,E2 14184.677} C_VEL
LIN {X 0,Y 421.277,Z 213.896,A -85,B 0,C 180,E1 14182.069,E2 14182.069} C_VEL
LIN {X 0,Y 430.961,Z 228.728,A -85,B 0,C 180,E1 14179.901,E2 14179.901} C_VEL
LIN {X 0,Y 436.348,Z 237.778,A -85,B 0,C 180,E1 14178.76,E2 14178.76} C_VEL
LIN {X 0,Y 438.076,Z 252.82,A -85,B 0,C 180,E1 14178.107,E2 14178.107} C_VEL
LIN {X 0,Y 429.957,Z 481.129,A -85,B 0,C 180,E1 14174.04,E2 14174.04} C_VEL
LIN {X 0,Y 428.444,Z 518.455,A -85,B 0,C 180,E1 14173.344,E2 14173.344} C_VEL
LIN {X 0,Y 426.596,Z 539.913,A -85,B 0,C 180,E1 14172.745,E2 14172.745} C_VEL
LIN {X 0,Y 424.182,Z 560.813,A -85,B 0,C 180,E1 14171.931,E2 14171.931} C_VEL
LIN {X 0,Y 421.307,Z 580.992,A -85,B 0,C 180,E1 14170.919,E2 14170.919} C_VEL
LIN {X 0,Y 417.936,Z 600.278,A -85,B 0,C 180,E1 14169.698,E2 14169.698} C_VEL
LIN {X 0,Y 414.069,Z 619.971,A -85,B 0,C 180,E1 14168.181,E2 14168.181} C_VEL
LIN {X 0,Y 410.149,Z 638.035,A -85,B 0,C 180,E1 14166.499,E2 14166.499} C_VEL
LIN {X 0,Y 406.078,Z 655.253,A -85,B 0,C 180,E1 14164.578,E2 14164.578} C_VEL
LIN {X 0,Y 405.508,Z 657.612,A -85,B 0,C 180,E1 14164.292,E2 14164.292} C_VEL
LIN {X 0,Y 403.258,Z 663.467,A -85,B 0,C 180,E1 14163.641,E2 14163.641} C_VEL
LIN {X 0,Y 394.474,Z 677.988,A -85,B 0,C 180,E1 14162.086,E2 14162.086} C_VEL
LIN {X 0,Y 392.212,Z 683.238,A -85,B 0,C 180,E1 14161.325,E2 14161.325} C_VEL
LIN {X 0,Y 388.421,Z 697.54,A -85,B 0,C 180,E1 14158.774,E2 14158.774} C_VEL
LIN {X 0,Y 385.004,Z 710.41,A -85,B 0,C 180,E1 14156.03,E2 14156.03} C_VEL
LIN {X 0,Y 381.988,Z 722.526,A -85,B 0,C 180,E1 14152.954,E2 14152.954} C_VEL
LIN {X 0,Y 379.713,Z 732.701,A -85,B 0,C 180,E1 14149.857,E2 14149.857} C_VEL
LIN {X 0,Y 378.077,Z 741.004,A -85,B 0,C 180,E1 14146.753,E2 14146.753} C_VEL
LIN {X 0,Y 376.933,Z 748.318,A -85,B 0,C 180,E1 14143.342,E2 14143.342} C_VEL
LIN {X 0,Y 376.33,Z 753.71,A -85,B 0,C 180,E1 14140.099,E2 14140.099} C_VEL
LIN {X 0,Y 376.057,Z 757.451,A -85,B 0,C 180,E1 14136.871,E2 14136.871} C_VEL
LIN {X 0,Y 375.956,Z 759.882,A -85,B 0,C 180,E1 14133.507,E2 14133.507} C_VEL
LIN {X 0,Y 375.932,Z 760.735,A -85,B 0,C 180,E1 14130.457,E2 14130.457} C_VEL
LIN {X 0,Y 375.947,Z 760.178,A -85,B 0,C 180,E1 14127.104,E2 14127.104} C_VEL
LIN {X 0,Y 376.021,Z 758.274,A -85,B 0,C 180,E1 14123.895,E2 14123.895} C_VEL
LIN {X 0,Y 376.228,Z 754.802,A -85,B 0,C 180,E1 14120.671,E2 14120.671} C_VEL
LIN {X 0,Y 376.766,Z 749.639,A -85,B 0,C 180,E1 14117.276,E2 14117.276} C_VEL
LIN {X 0,Y 377.74,Z 743.064,A -85,B 0,C 180,E1 14114.022,E2 14114.022} C_VEL
LIN {X 0,Y 379.282,Z 734.702,A -85,B 0,C 180,E1 14110.761,E2 14110.761} C_VEL
LIN {X 0,Y 381.538,Z 724.483,A -85,B 0,C 180,E1 14107.505,E2 14107.505} C_VEL
LIN {X 0,Y 384.43,Z 712.789,A -85,B 0,C 180,E1 14104.422,E2 14104.422} C_VEL
LIN {X 0,Y 387.688,Z 700.185,A -85,B 0,C 180,E1 14101.671,E2 14101.671} C_VEL
LIN {X 0,Y 391.624,Z 685.475,A -85,B 0,C 180,E1 14098.955,E2 14098.955} C_VEL
LIN {X 0,Y 395.727,Z 670.265,A -85,B 0,C 180,E1 14096.579,E2 14096.579} C_VEL
LIN {X 0,Y 399.895,Z 654.033,A -85,B 0,C 180,E1 14094.458,E2 14094.458} C_VEL
LIN {X 0,Y 404.279,Z 636.089,A -85,B 0,C 180,E1 14092.475,E2 14092.475} C_VEL
LIN {X 0,Y 408.533,Z 617.441,A -85,B 0,C 180,E1 14090.755,E2 14090.755} C_VEL
LIN {X 0,Y 412.406,Z 598.075,A -85,B 0,C 180,E1 14089.295,E2 14089.295} C_VEL
LIN {X 0,Y 416.107,Z 576.861,A -85,B 0,C 180,E1 14087.996,E2 14087.996} C_VEL
LIN {X 0,Y 419.148,Z 555.965,A -85,B 0,C 180,E1 14086.983,E2 14086.983} C_VEL
LIN {X 0,Y 421.531,Z 534.603,A -85,B 0,C 180,E1 14086.217,E2 14086.217} C_VEL
LIN {X 0,Y 423.333,Z 511.453,A -85,B 0,C 180,E1 14085.637,E2 14085.637} C_VEL
LIN {X 0,Y 431.653,Z 288.017,A -85,B 0,C 180,E1 14081.616,E2 14081.616} C_VEL
LIN {X 0,Y 432.954,Z 252.453,A -85,B 0,C 180,E1 14080.942,E2 14080.942} C_VEL
LIN {X 0,Y 431.526,Z 241.74,A -85,B 0,C 180,E1 14080.427,E2 14080.427} C_VEL
LIN {X 0,Y 421.039,Z 224.944,A -85,B 0,C 180,E1 14078.086,E2 14078.086} C_VEL
LIN {X 0,Y 411.164,Z 210.23,A -85,B 0,C 180,E1 14075.663,E2 14075.663} C_VEL
LIN {X 0,Y 403.112,Z 199.102,A -85,B 0,C 180,E1 14073.496,E2 14073.496} C_VEL
LIN {X 0,Y 401.053,Z 195.665,A -85,B 0,C 180,E1 14072.752,E2 14072.752} C_VEL
LIN {X 0,Y 395.33,Z 185.261,A -85,B 0,C 180,E1 14069.717,E2 14069.717} C_VEL
LIN {X 0,Y 392.791,Z 180.757,A -85,B 0,C 180,E1 14068.26,E2 14068.26} C_VEL
LIN {X 0,Y 390.425,Z 176.417,A -85,B 0,C 180,E1 14066.791,E2 14066.791} C_VEL
LIN {X 0,Y 387.928,Z 172.038,A -85,B 0,C 180,E1 14065.168,E2 14065.168} C_VEL
LIN {X 0,Y 385.03,Z 167.579,A -85,B 0,C 180,E1 14063.249,E2 14063.249} C_VEL
LIN {X 0,Y 384.324,Z 166.01,A -85,B 0,C 180,E1 14062.646,E2 14062.646} C_VEL
LIN {X 0,Y 381.965,Z 162.958,A -85,B 0,C 180,E1 14061.016,E2 14061.016} C_VEL
LIN {X 0,Y 380.884,Z 160.501,A -85,B 0,C 180,E1 14059.954,E2 14059.954} C_VEL
LIN {X 0,Y 378.139,Z 156.941,A -85,B 0,C 180,E1 14057.703,E2 14057.703} C_VEL
LIN {X 0,Y 377.703,Z 155.209,A -85,B 0,C 180,E1 14056.771,E2 14056.771} C_VEL
LIN {X 0,Y 377.674,Z 155,A -85,B 0,C 180,E1 14052.849,E2 14052.849} C_VEL
LIN {X 0,Y 377.682,Z 154.997,A -85,B 0,C 180,E1 14048.679,E2 14048.679} C_VEL
LIN {X 0,Y 377.678,Z 154.99,A -85,B 0,C 180,E1 14044.708,E2 14044.708} C_VEL
LIN {X 0,Y 377.688,Z 154.984,A -85,B 0,C 180,E1 14040.607,E2 14040.607} C_VEL
LIN {X 0,Y 377.676,Z 154.985,A -85,B 0,C 180,E1 14036.509,E2 14036.509} C_VEL
LIN {X 0,Y 377.678,Z 154.987,A -85,B 0,C 180,E1 14032.394,E2 14032.394} C_VEL
LIN {X 0,Y 377.676,Z 154.994,A -85,B 0,C 180,E1 14028.381,E2 14028.381} C_VEL
LIN {X 0,Y 377.693,Z 155.219,A -85,B 0,C 180,E1 14025.591,E2 14025.591} C_VEL
LIN {X 0,Y 379.631,Z 159.279,A -85,B 0,C 180,E1 14023.317,E2 14023.317} C_VEL
LIN {X 0,Y 381.466,Z 161.349,A -85,B 0,C 180,E1 14021.984,E2 14021.984} C_VEL
LIN {X 0,Y 383.404,Z 165.058,A -85,B 0,C 180,E1 14020.342,E2 14020.342} C_VEL
LIN {X 0,Y 385.007,Z 166.999,A -85,B 0,C 180,E1 14019.318,E2 14019.318} C_VEL
LIN {X 0,Y 387.036,Z 170.747,A -85,B 0,C 180,E1 14017.842,E2 14017.842} C_VEL
LIN {X 0,Y 388.252,Z 172.403,A -85,B 0,C 180,E1 14017.116,E2 14017.116} C_VEL
LIN {X 0,Y 390.183,Z 175.854,A -85,B 0,C 180,E1 14015.956,E2 14015.956} C_VEL
LIN {X 0,Y 392.377,Z 178.276,A -85,B 0,C 180,E1 14015.217,E2 14015.217} C_VEL
LIN {X 0,Y 397.369,Z 184.249,A -85,B 0,C 180,E1 14013.634,E2 14013.634} C_VEL
LIN {X 0,Y 402.046,Z 190.013,A -85,B 0,C 180,E1 14012.246,E2 14012.246} C_VEL
LIN {X 0,Y 406.794,Z 196.016,A -85,B 0,C 180,E1 14010.919,E2 14010.919} C_VEL
LIN {X 0,Y 413.63,Z 204.895,A -85,B 0,C 180,E1 14009.132,E2 14009.132} C_VEL
LIN {X 0,Y 424.044,Z 219.362,A -85,B 0,C 180,E1 14006.634,E2 14006.634} C_VEL
LIN {X 0,Y 435.132,Z 236.192,A -85,B 0,C 180,E1 14004.212,E2 14004.212} C_VEL
LIN {X 0,Y 436.751,Z 239.091,A -85,B 0,C 180,E1 14003.867,E2 14003.867} C_VEL
LIN {X 0,Y 427.218,Z 450.476,A -85,B 0,C 180,E1 13999.793,E2 13999.793} C_VEL
LIN {X 0,Y 424.31,Z 512.849,A -85,B 0,C 180,E1 13998.557,E2 13998.557} C_VEL
LIN {X 0,Y 422.1,Z 536.177,A -85,B 0,C 180,E1 13997.891,E2 13997.891} C_VEL
LIN {X 0,Y 419.14,Z 560.526,A -85,B 0,C 180,E1 13996.932,E2 13996.932} C_VEL
LIN {X 0,Y 416.063,Z 581.304,A -85,B 0,C 180,E1 13995.878,E2 13995.878} C_VEL
LIN {X 0,Y 412.351,Z 602.711,A -85,B 0,C 180,E1 13994.53,E2 13994.53} C_VEL
LIN {X 0,Y 408.597,Z 622.292,A -85,B 0,C 180,E1 13993.056,E2 13993.056} C_VEL
LIN {X 0,Y 404.376,Z 642.109,A -85,B 0,C 180,E1 13991.265,E2 13991.265} C_VEL
LIN {X 0,Y 400.076,Z 661.409,A -85,B 0,C 180,E1 13989.218,E2 13989.218} C_VEL
LIN {X 0,Y 395.993,Z 678.899,A -85,B 0,C 180,E1 13987.026,E2 13987.026} C_VEL
LIN {X 0,Y 391.643,Z 697.226,A -85,B 0,C 180,E1 13984.346,E2 13984.346} C_VEL
LIN {X 0,Y 388.063,Z 712.699,A -85,B 0,C 180,E1 13981.709,E2 13981.709} C_VEL
LIN {X 0,Y 384.839,Z 726.822,A -85,B 0,C 180,E1 13978.888,E2 13978.888} C_VEL
LIN {X 0,Y 382.051,Z 740.176,A -85,B 0,C 180,E1 13975.806,E2 13975.806} C_VEL
LIN {X 0,Y 379.924,Z 751.358,A -85,B 0,C 180,E1 13972.759,E2 13972.759} C_VEL
LIN {X 0,Y 378.166,Z 762.078,A -85,B 0,C 180,E1 13969.284,E2 13969.284} C_VEL
LIN {X 0,Y 377.147,Z 769.61,A -85,B 0,C 180,E1 13966.32,E2 13966.32} C_VEL
LIN {X 0,Y 376.41,Z 776.905,A -85,B 0,C 180,E1 13962.736,E2 13962.736} C_VEL
LIN {X 0,Y 376.088,Z 781.485,A -85,B 0,C 180,E1 13959.796,E2 13959.796} C_VEL
LIN {X 0,Y 375.954,Z 785.287,A -85,B 0,C 180,E1 13956.413,E2 13956.413} C_VEL
LIN {X 0,Y 375.922,Z 787.292,A -85,B 0,C 180,E1 13953.354,E2 13953.354} C_VEL
LIN {X 0,Y 375.923,Z 788.125,A -85,B 0,C 180,E1 13950.152,E2 13950.152} C_VEL
LIN {X 0,Y 375.924,Z 787.434,A -85,B 0,C 180,E1 13946.951,E2 13946.951} C_VEL
LIN {X 0,Y 375.939,Z 785.642,A -85,B 0,C 180,E1 13944.046,E2 13944.046} C_VEL
LIN {X 0,Y 376.062,Z 782.133,A -85,B 0,C 180,E1 13940.667,E2 13940.667} C_VEL
LIN {X 0,Y 376.368,Z 777.446,A -85,B 0,C 180,E1 13937.574,E2 13937.574} C_VEL
LIN {X 0,Y 376.984,Z 771.094,A -85,B 0,C 180,E1 13934.305,E2 13934.305} C_VEL
LIN {X 0,Y 378.041,Z 762.911,A -85,B 0,C 180,E1 13931.016,E2 13931.016} C_VEL
LIN {X 0,Y 379.645,Z 752.998,A -85,B 0,C 180,E1 13927.714,E2 13927.714} C_VEL
LIN {X 0,Y 381.685,Z 741.95,A -85,B 0,C 180,E1 13924.656,E2 13924.656} C_VEL
LIN {X 0,Y 384.535,Z 728.249,A -85,B 0,C 180,E1 13921.418,E2 13921.418} C_VEL
LIN {X 0,Y 387.664,Z 714.358,A -85,B 0,C 180,E1 13918.602,E2 13918.602} C_VEL
LIN {X 0,Y 391.307,Z 698.631,A -85,B 0,C 180,E1 13915.881,E2 13915.881} C_VEL
LIN {X 0,Y 395.333,Z 681.752,A -85,B 0,C 180,E1 13913.354,E2 13913.354} C_VEL
LIN {X 0,Y 399.394,Z 664.282,A -85,B 0,C 180,E1 13911.129,E2 13911.129} C_VEL
LIN {X 0,Y 403.958,Z 643.954,A -85,B 0,C 180,E1 13908.918,E2 13908.918} C_VEL
LIN {X 0,Y 408.267,Z 623.863,A -85,B 0,C 180,E1 13907.076,E2 13907.076} C_VEL
LIN {X 0,Y 412.066,Z 604.143,A -85,B 0,C 180,E1 13905.572,E2 13905.572} C_VEL
LIN {X 0,Y 415.781,Z 583.117,A -85,B 0,C 180,E1 13904.225,E2 13904.225} C_VEL
LIN {X 0,Y 418.926,Z 561.926,A -85,B 0,C 180,E1 13903.137,E2 13903.137} C_VEL
LIN {X 0,Y 421.801,Z 538.944,A -85,B 0,C 180,E1 13902.205,E2 13902.205} C_VEL
LIN {X 0,Y 423.936,Z 516.739,A -85,B 0,C 180,E1 13901.545,E2 13901.545} C_VEL
LIN {X 0,Y 425.716,Z 484.599,A -85,B 0,C 180,E1 13900.87,E2 13900.87} C_VEL
LIN {X 0,Y 435.034,Z 275.902,A -85,B 0,C 180,E1 13896.844,E2 13896.844} C_VEL
LIN {X 0,Y 436.637,Z 238.611,A -85,B 0,C 180,E1 13896.112,E2 13896.112} C_VEL
LIN {X 0,Y 425.583,Z 221.61,A -85,B 0,C 180,E1 13893.727,E2 13893.727} C_VEL
LIN {X 0,Y 415.753,Z 207.826,A -85,B 0,C 180,E1 13891.417,E2 13891.417} C_VEL
LIN {X 0,Y 407.767,Z 197.263,A -85,B 0,C 180,E1 13889.367,E2 13889.367} C_VEL
LIN {X 0,Y 403.53,Z 191.926,A -85,B 0,C 180,E1 13888.205,E2 13888.205} C_VEL
LIN {X 0,Y 399.656,Z 187.049,A -85,B 0,C 180,E1 13887.086,E2 13887.086} C_VEL
